SPLINE
SPL {X  -159.452, Y  +378.767, Z    +0.000, E1   +11.887, E3 +105762.657}
SPL {X  -159.840, Y  +384.856, Z    +0.000, E1    +7.126, E3 +105781.629}
SPL {X  -159.991, Y  +390.336, Z    +0.000, E1    +2.803, E3 +105795.451}
SPL {X  -160.000, Y  +403.532, Z    +0.000, E1    -6.523, E3 +105813.172}
SPL {X  -160.000, Y  +409.023, Z    +0.000, E1   -10.003, E3 +105823.946}
SPL {X  -160.000, Y  +418.032, Z    +0.000, E1   -14.569, E3 +105848.805}
SPL {X  -160.000, Y  +420.561, Z    +0.000, E1   -14.816, E3 +105866.285}
SPL {X  -160.000, Y  +422.801, Z    +0.000, E1   -14.823, E3 +105884.233}
SPL {X  -160.000, Y  +425.518, Z    +0.000, E1   -14.845, E3 +105906.008}
SPL {X  -160.000, Y  +428.688, Z    +0.000, E1   -14.854, E3 +105931.416}
SPL {X  -160.000, Y  +431.971, Z    +0.000, E1   -14.849, E3 +105957.885}
SPL {X  -160.000, Y  +435.345, Z    +0.000, E1   -14.857, E3 +105984.935}
SPL {X  -160.000, Y  +438.732, Z    +0.000, E1   -14.858, E3 +106012.083}
SPL {X  -160.000, Y  +441.925, Z    +0.000, E1   -14.848, E3 +106037.754}
SPL {X  -160.000, Y  +444.299, Z    +0.000, E1   -14.809, E3 +106056.938}
SPL {X  -160.000, Y  +446.229, Z    +0.000, E1   -14.820, E3 +106072.357}
SPL {X  -160.000, Y  +448.987, Z    +0.000, E1   -14.868, E3 +106094.294}
SPL {X  -160.000, Y  +452.351, Z    +0.000, E1   -14.871, E3 +106121.270}
SPL {X  -160.000, Y  +455.709, Z    +0.000, E1   -14.880, E3 +106148.084}
SPL {X  -160.000, Y  +458.189, Z    +0.000, E1   -14.832, E3 +106168.086}
SPL {X  -160.000, Y  +459.885, Z    +0.000, E1   -14.825, E3 +106181.757}
SPL {X  -160.000, Y  +462.438, Z    +0.000, E1   -14.868, E3 +106202.167}
SPL {X  -160.000, Y  +465.575, Z    +0.000, E1   -14.849, E3 +106227.475}
SPL {X  -160.000, Y  +468.581, Z    +0.000, E1   -14.841, E3 +106251.707}
SPL {X  -160.000, Y  +471.795, Z    +0.000, E1   -14.854, E3 +106277.495}
SPL {X  -160.000, Y  +475.138, Z    +0.000, E1   -14.853, E3 +106304.345}
SPL {X  -160.000, Y  +477.981, Z    +0.000, E1   -14.823, E3 +106327.265}
SPL {X  -160.000, Y  +480.658, Z    +0.000, E1   -14.835, E3 +106348.741}
SPL {X  -160.000, Y  +483.534, Z    +0.000, E1   -14.838, E3 +106371.836}
SPL {X  -160.000, Y  +486.226, Z    +0.000, E1   -14.823, E3 +106393.501}
SPL {X  -160.000, Y  +488.751, Z    +0.000, E1   -14.827, E3 +106413.774}
SPL {X  -160.000, Y  +491.612, Z    +0.000, E1   -14.844, E3 +106436.696}
SPL {X  -160.000, Y  +494.417, Z    +0.000, E1   -14.827, E3 +106459.287}
SPL {X  -160.000, Y  +496.961, Z    +0.000, E1   -14.824, E3 +106479.731}
SPL {X  -160.000, Y  +499.610, Z    +0.000, E1   -14.830, E3 +106501.004}
SPL {X  -160.000, Y  +502.268, Z    +0.000, E1   -14.832, E3 +106522.273}
SPL {X  -160.000, Y  +505.041, Z    +0.000, E1   -14.849, E3 +106544.435}
SPL {X  -160.000, Y  +507.743, Z    +0.000, E1   -14.842, E3 +106566.059}
SPL {X  -160.000, Y  +510.437, Z    +0.000, E1   -14.860, E3 +106587.573}
SPL {X  -160.000, Y  +513.179, Z    +0.000, E1   -14.849, E3 +106609.620}
SPL {X  -160.000, Y  +515.613, Z    +0.000, E1   -14.829, E3 +106629.291}
SPL {X  -160.000, Y  +518.188, Z    +0.000, E1   -14.845, E3 +106649.920}
SPL {X  -160.000, Y  +520.790, Z    +0.000, E1   -14.839, E3 +106670.749}
SPL {X  -160.000, Y  +523.469, Z    +0.000, E1   -14.855, E3 +106692.197}
SPL {X  -160.000, Y  +526.403, Z    +0.000, E1   -14.858, E3 +106715.734}
SPL {X  -160.000, Y  +529.266, Z    +0.000, E1   -14.848, E3 +106738.741}
SPL {X  -160.000, Y  +531.688, Z    +0.000, E1   -14.826, E3 +106758.291}
SPL {X  -160.000, Y  +534.214, Z    +0.000, E1   -14.841, E3 +106778.554}
SPL {X  -160.000, Y  +537.002, Z    +0.000, E1   -14.839, E3 +106800.972}
SPL {X  -160.000, Y  +539.729, Z    +0.000, E1   -14.840, E3 +106822.783}
SPL {X  -160.000, Y  +542.408, Z    +0.000, E1   -14.839, E3 +106844.336}
SPL {X  -160.000, Y  +545.014, Z    +0.000, E1   -14.831, E3 +106865.282}
SPL {X  -160.000, Y  +547.659, Z    +0.000, E1   -14.839, E3 +106886.496}
SPL {X  -160.000, Y  +550.215, Z    +0.000, E1   -14.827, E3 +106907.061}
SPL {X  -160.000, Y  +552.762, Z    +0.000, E1   -14.836, E3 +106927.479}
SPL {X  -160.000, Y  +555.331, Z    +0.000, E1   -14.837, E3 +106948.020}
SPL {X  -160.000, Y  +558.235, Z    +0.000, E1   -14.869, E3 +106971.184}
SPL {X  -160.000, Y  +561.088, Z    +0.000, E1   -14.848, E3 +106994.102}
SPL {X  -160.000, Y  +563.693, Z    +0.000, E1   -14.852, E3 +107014.963}
SPL {X  -160.000, Y  +566.560, Z    +0.000, E1   -14.865, E3 +107037.941}
SPL {X  -160.000, Y  +569.305, Z    +0.000, E1   -14.848, E3 +107059.969}
SPL {X  -160.000, Y  +571.769, Z    +0.000, E1   -14.852, E3 +107079.715}
SPL {X  -160.000, Y  +574.366, Z    +0.000, E1   -14.855, E3 +107100.502}
SPL {X  -160.000, Y  +577.037, Z    +0.000, E1   -14.859, E3 +107121.901}
SPL {X  -160.000, Y  +579.855, Z    +0.000, E1   -14.869, E3 +107144.429}
SPL {X  -160.000, Y  +582.456, Z    +0.000, E1   -14.854, E3 +107165.289}
SPL {X  -160.000, Y  +585.083, Z    +0.000, E1   -14.866, E3 +107186.338}
SPL {X  -160.000, Y  +587.675, Z    +0.000, E1   -14.853, E3 +107207.129}
SPL {X  -160.000, Y  +590.216, Z    +0.000, E1   -14.864, E3 +107227.448}
SPL {X  -160.000, Y  +592.848, Z    +0.000, E1   -14.865, E3 +107248.500}
SPL {X  -160.000, Y  +595.342, Z    +0.000, E1   -14.848, E3 +107268.677}
SPL {X  -160.000, Y  +597.995, Z    +0.000, E1   -14.848, E3 +107290.017}
SPL {X  -160.000, Y  +600.731, Z    +0.000, E1   -14.846, E3 +107311.969}
SPL {X  -160.000, Y  +603.404, Z    +0.000, E1   -14.846, E3 +107333.404}
SPL {X  -160.000, Y  +605.923, Z    +0.000, E1   -14.838, E3 +107353.645}
SPL {X  -160.000, Y  +608.492, Z    +0.000, E1   -14.846, E3 +107374.249}
SPL {X  -160.000, Y  +611.345, Z    +0.000, E1   -14.856, E3 +107397.107}
SPL {X  -160.000, Y  +614.087, Z    +0.000, E1   -14.839, E3 +107419.166}
SPL {X  -160.000, Y  +616.566, Z    +0.000, E1   -14.839, E3 +107439.060}
SPL {X  -160.000, Y  +619.350, Z    +0.000, E1   -14.855, E3 +107461.348}
SPL {X  -160.000, Y  +622.198, Z    +0.000, E1   -14.846, E3 +107484.233}
SPL {X  -160.000, Y  +624.642, Z    +0.000, E1   -14.829, E3 +107503.905}
SPL {X  -160.000, Y  +627.119, Z    +0.000, E1   -14.843, E3 +107523.745}
SPL {X  -160.000, Y  +629.682, Z    +0.000, E1   -14.838, E3 +107544.314}
SPL {X  -160.000, Y  +632.223, Z    +0.000, E1   -14.841, E3 +107564.705}
SPL {X  -160.000, Y  +634.941, Z    +0.000, E1   -14.846, E3 +107586.503}
SPL {X  -160.000, Y  +637.723, Z    +0.000, E1   -14.844, E3 +107608.847}
SPL {X  -160.000, Y  +640.315, Z    +0.000, E1   -14.836, E3 +107629.645}
SPL {X  -160.000, Y  +643.085, Z    +0.000, E1   -14.865, E3 +107651.696}
SPL {X  -160.000, Y  +645.845, Z    +0.000, E1   -14.848, E3 +107673.884}
SPL {X  -160.000, Y  +648.229, Z    +0.000, E1   -14.834, E3 +107693.094}
SPL {X  -160.000, Y  +650.656, Z    +0.000, E1   -14.835, E3 +107712.651}
SPL {X  -160.000, Y  +653.134, Z    +0.000, E1   -14.827, E3 +107732.578}
SPL {X  -160.000, Y  +655.670, Z    +0.000, E1   -14.841, E3 +107752.872}
SPL {X  -160.000, Y  +658.349, Z    +0.000, E1   -14.842, E3 +107774.347}
SPL {X  -160.000, Y  +660.936, Z    +0.000, E1   -14.838, E3 +107795.099}
SPL {X  -160.000, Y  +663.567, Z    +0.000, E1   -14.845, E3 +107816.230}
SPL {X  -160.000, Y  +666.216, Z    +0.000, E1   -14.832, E3 +107837.546}
SPL {X  -159.997, Y  +668.731, Z    +0.000, E1   -14.834, E3 +107857.738}
SPL {X  -159.962, Y  +671.176, Z    +0.000, E1   -14.822, E3 +107877.449}
SPL {X  -159.895, Y  +673.507, Z    +0.000, E1   -14.821, E3 +107896.181}
SPL {X  -159.785, Y  +675.985, Z    +0.000, E1   -14.818, E3 +107916.182}
SPL {X  -159.627, Y  +678.622, Z    +0.000, E1   -14.804, E3 +107937.535}
SPL {X  -159.438, Y  +681.094, Z    +0.000, E1   -14.770, E3 +107957.706}
SPL {X  -159.262, Y  +683.054, Z    +0.000, E1   -14.719, E3 +107973.935}
ENDSPLINE

SPLINE
SPL {X  -159.661, Y  +678.114, Z    +0.000, E1    -9.575, E3 +108003.527}
SPL {X  -159.942, Y  +672.020, Z    +0.000, E1    -4.692, E3 +108022.153}
SPL {X  -160.000, Y  +664.971, Z    +0.000, E1    +0.516, E3 +108041.704}
SPL {X  -160.000, Y  +660.032, Z    +0.000, E1    +3.995, E3 +108053.647}
SPL {X  -160.000, Y  +652.280, Z    +0.000, E1    +8.913, E3 +108072.162}
SPL {X  -160.000, Y  +644.147, Z    +0.000, E1   +13.158, E3 +108095.712}
SPL {X  -160.000, Y  +641.594, Z    +0.000, E1   +13.488, E3 +108114.153}
SPL {X  -160.000, Y  +639.799, Z    +0.000, E1   +13.486, E3 +108130.063}
SPL {X  -160.000, Y  +637.896, Z    +0.000, E1   +13.493, E3 +108146.878}
SPL {X  -160.000, Y  +635.832, Z    +0.000, E1   +13.499, E3 +108165.137}
SPL {X  -160.000, Y  +633.839, Z    +0.000, E1   +13.489, E3 +108182.826}
SPL {X  -160.000, Y  +631.625, Z    +0.000, E1   +13.508, E3 +108202.366}
SPL {X  -160.000, Y  +629.417, Z    +0.000, E1   +13.491, E3 +108221.978}
SPL {X  -160.000, Y  +627.180, Z    +0.000, E1   +13.508, E3 +108241.732}
SPL {X  -160.000, Y  +624.970, Z    +0.000, E1   +13.490, E3 +108261.382}
SPL {X  -160.000, Y  +623.020, Z    +0.000, E1   +13.491, E3 +108278.612}
SPL {X  -160.000, Y  +620.888, Z    +0.000, E1   +13.501, E3 +108297.474}
SPL {X  -160.000, Y  +618.790, Z    +0.000, E1   +13.488, E3 +108316.096}
SPL {X  -160.000, Y  +616.631, Z    +0.000, E1   +13.504, E3 +108335.150}
SPL {X  -160.000, Y  +614.230, Z    +0.000, E1   +13.510, E3 +108356.346}
SPL {X  -160.000, Y  +612.132, Z    +0.000, E1   +13.485, E3 +108375.062}
SPL {X  -160.000, Y  +610.405, Z    +0.000, E1   +13.477, E3 +108390.436}
SPL {X  -160.000, Y  +608.437, Z    +0.000, E1   +13.502, E3 +108407.691}
SPL {X  -160.000, Y  +606.281, Z    +0.000, E1   +13.502, E3 +108426.709}
SPL {X  -160.000, Y  +604.124, Z    +0.000, E1   +13.513, E3 +108445.764}
SPL {X  -160.000, Y  +601.878, Z    +0.000, E1   +13.505, E3 +108465.661}
SPL {X  -160.000, Y  +599.648, Z    +0.000, E1   +13.506, E3 +108485.438}
SPL {X  -160.000, Y  +597.673, Z    +0.000, E1   +13.479, E3 +108503.111}
SPL {X  -160.000, Y  +595.601, Z    +0.000, E1   +13.499, E3 +108521.395}
SPL {X  -160.000, Y  +593.187, Z    +0.000, E1   +13.500, E3 +108542.775}
SPL {X  -160.000, Y  +591.079, Z    +0.000, E1   +13.483, E3 +108561.501}
SPL {X  -160.000, Y  +589.151, Z    +0.000, E1   +13.489, E3 +108578.552}
SPL {X  -160.000, Y  +586.908, Z    +0.000, E1   +13.501, E3 +108598.397}
SPL {X  -160.000, Y  +584.660, Z    +0.000, E1   +13.490, E3 +108618.339}
SPL {X  -160.000, Y  +582.409, Z    +0.000, E1   +13.499, E3 +108638.257}
SPL {X  -160.000, Y  +580.150, Z    +0.000, E1   +13.490, E3 +108658.304}
SPL {X  -160.000, Y  +577.953, Z    +0.000, E1   +13.493, E3 +108677.762}
SPL {X  -160.000, Y  +575.630, Z    +0.000, E1   +13.502, E3 +108698.246}
SPL {X  -160.000, Y  +573.418, Z    +0.000, E1   +13.502, E3 +108717.754}
SPL {X  -160.000, Y  +571.226, Z    +0.000, E1   +13.520, E3 +108736.963}
SPL {X  -160.000, Y  +569.166, Z    +0.000, E1   +13.512, E3 +108755.153}
SPL {X  -160.000, Y  +567.275, Z    +0.000, E1   +13.517, E3 +108771.820}
SPL {X  -160.000, Y  +565.259, Z    +0.000, E1   +13.523, E3 +108789.609}
SPL {X  -160.000, Y  +563.305, Z    +0.000, E1   +13.512, E3 +108806.948}
SPL {X  -160.000, Y  +561.240, Z    +0.000, E1   +13.521, E3 +108825.209}
SPL {X  -160.000, Y  +558.881, Z    +0.000, E1   +13.524, E3 +108846.052}
SPL {X  -160.000, Y  +556.697, Z    +0.000, E1   +13.510, E3 +108865.438}
SPL {X  -160.000, Y  +554.624, Z    +0.000, E1   +13.512, E3 +108883.769}
SPL {X  -160.000, Y  +552.465, Z    +0.000, E1   +13.514, E3 +108902.853}
SPL {X  -160.000, Y  +550.315, Z    +0.000, E1   +13.514, E3 +108921.846}
SPL {X  -160.000, Y  +548.056, Z    +0.000, E1   +13.519, E3 +108941.847}
SPL {X  -160.000, Y  +545.826, Z    +0.000, E1   +13.501, E3 +108961.725}
SPL {X  -160.000, Y  +543.677, Z    +0.000, E1   +13.502, E3 +108980.783}
SPL {X  -160.000, Y  +541.664, Z    +0.000, E1   +13.489, E3 +108998.668}
SPL {X  -160.000, Y  +539.659, Z    +0.000, E1   +13.494, E3 +109016.429}
SPL {X  -160.000, Y  +537.370, Z    +0.000, E1   +13.501, E3 +109036.668}
SPL {X  -160.000, Y  +535.056, Z    +0.000, E1   +13.506, E3 +109057.063}
SPL {X  -160.000, Y  +532.975, Z    +0.000, E1   +13.494, E3 +109075.550}
SPL {X  -160.000, Y  +530.925, Z    +0.000, E1   +13.499, E3 +109093.712}
SPL {X  -160.000, Y  +528.768, Z    +0.000, E1   +13.498, E3 +109112.813}
SPL {X  -160.000, Y  +526.547, Z    +0.000, E1   +13.499, E3 +109132.482}
SPL {X  -160.000, Y  +523.964, Z    +0.000, E1   +13.742, E3 +109151.986}
SPL {X  -160.000, Y  +513.971, Z    +0.000, E1   +18.644, E3 +109170.898}
SPL {X  -160.000, Y  +513.562, Z    +0.000, E1   +16.972, E3 +109190.775}
SPL {X  -160.000, Y  +513.358, Z    +0.000, E1   +15.267, E3 +109211.047}
SPL {X  -160.000, Y  +512.244, Z    +0.000, E1   +14.473, E3 +109229.503}
SPL {X  -160.000, Y  +509.675, Z    +0.000, E1   +14.481, E3 +109250.647}
SPL {X  -160.000, Y  +507.162, Z    +0.000, E1   +14.470, E3 +109271.387}
SPL {X  -160.000, Y  +504.735, Z    +0.000, E1   +14.473, E3 +109291.358}
SPL {X  -160.000, Y  +502.261, Z    +0.000, E1   +14.476, E3 +109311.694}
SPL {X  -160.000, Y  +499.798, Z    +0.000, E1   +14.482, E3 +109331.896}
SPL {X  -160.000, Y  +497.435, Z    +0.000, E1   +14.476, E3 +109351.373}
SPL {X  -160.000, Y  +495.089, Z    +0.000, E1   +14.475, E3 +109370.740}
SPL {X  -160.000, Y  +492.764, Z    +0.000, E1   +14.469, E3 +109389.911}
SPL {X  -160.000, Y  +490.292, Z    +0.000, E1   +14.476, E3 +109410.312}
SPL {X  -160.000, Y  +487.641, Z    +0.000, E1   +14.470, E3 +109432.208}
SPL {X  -160.000, Y  +485.054, Z    +0.000, E1   +14.460, E3 +109453.651}
SPL {X  -160.000, Y  +482.421, Z    +0.000, E1   +14.461, E3 +109475.369}
SPL {X  -160.000, Y  +480.000, Z    +0.000, E1   +14.451, E3 +109495.334}
SPL {X  -160.000, Y  +477.551, Z    +0.000, E1   +14.466, E3 +109515.462}
SPL {X  -160.000, Y  +475.253, Z    +0.000, E1   +14.450, E3 +109534.436}
SPL {X  -160.000, Y  +473.070, Z    +0.000, E1   +14.454, E3 +109552.457}
SPL {X  -160.000, Y  +470.603, Z    +0.000, E1   +14.464, E3 +109572.757}
SPL {X  -160.000, Y  +468.243, Z    +0.000, E1   +14.458, E3 +109592.157}
SPL {X  -160.000, Y  +465.791, Z    +0.000, E1   +14.475, E3 +109612.301}
SPL {X  -160.000, Y  +463.103, Z    +0.000, E1   +14.474, E3 +109634.449}
SPL {X  -160.000, Y  +460.743, Z    +0.000, E1   +14.465, E3 +109653.858}
SPL {X  -160.000, Y  +458.292, Z    +0.000, E1   +14.492, E3 +109673.857}
SPL {X  -160.000, Y  +455.874, Z    +0.000, E1   +14.484, E3 +109693.715}
SPL {X  -160.000, Y  +453.555, Z    +0.000, E1   +14.488, E3 +109712.794}
SPL {X  -160.000, Y  +451.093, Z    +0.000, E1   +14.485, E3 +109733.106}
SPL {X  -160.000, Y  +448.700, Z    +0.000, E1   +14.483, E3 +109752.795}
SPL {X  -160.000, Y  +446.277, Z    +0.000, E1   +14.485, E3 +109772.719}
SPL {X  -160.000, Y  +443.879, Z    +0.000, E1   +14.485, E3 +109792.457}
SPL {X  -160.000, Y  +441.447, Z    +0.000, E1   +14.485, E3 +109812.464}
SPL {X  -160.000, Y  +439.006, Z    +0.000, E1   +14.488, E3 +109832.547}
SPL {X  -160.000, Y  +436.311, Z    +0.000, E1   +14.498, E3 +109854.706}
SPL {X  -160.000, Y  +433.559, Z    +0.000, E1   +14.491, E3 +109877.376}
SPL {X  -160.000, Y  +431.162, Z    +0.000, E1   +14.479, E3 +109897.127}
SPL {X  -160.000, Y  +429.152, Z    +0.000, E1   +14.469, E3 +109913.708}
SPL {X  -160.000, Y  +426.863, Z    +0.000, E1   +14.490, E3 +109932.487}
SPL {X  -160.000, Y  +424.653, Z    +0.000, E1   +14.467, E3 +109950.747}
SPL {X  -160.000, Y  +422.337, Z    +0.000, E1   +14.492, E3 +109969.731}
SPL {X  -160.000, Y  +419.639, Z    +0.000, E1   +14.504, E3 +109991.771}
SPL {X  -160.000, Y  +417.127, Z    +0.000, E1   +14.501, E3 +110012.362}
SPL {X  -160.000, Y  +414.849, Z    +0.000, E1   +14.496, E3 +110031.096}
SPL {X  -160.000, Y  +412.396, Z    +0.000, E1   +14.505, E3 +110051.285}
SPL {X  -160.000, Y  +409.815, Z    +0.000, E1   +14.498, E3 +110072.539}
SPL {X  -160.000, Y  +407.614, Z    +0.000, E1   +14.484, E3 +110090.665}
SPL {X  -160.000, Y  +405.406, Z    +0.000, E1   +14.501, E3 +110108.728}
SPL {X  -160.000, Y  +402.958, Z    +0.000, E1   +14.500, E3 +110128.898}
SPL {X  -160.000, Y  +400.690, Z    +0.000, E1   +14.484, E3 +110147.609}
SPL {X  -160.000, Y  +398.391, Z    +0.000, E1   +14.502, E3 +110166.435}
SPL {X  -160.000, Y  +395.999, Z    +0.000, E1   +14.484, E3 +110186.225}
SPL {X  -160.000, Y  +393.685, Z    +0.000, E1   +14.486, E3 +110205.298}
SPL {X  -159.999, Y  +391.313, Z    +0.000, E1   +14.479, E3 +110224.880}
SPL {X  -159.970, Y  +388.900, Z    +0.000, E1   +14.480, E3 +110244.764}
SPL {X  -159.903, Y  +386.417, Z    +0.000, E1   +14.475, E3 +110265.269}
SPL {X  -159.796, Y  +383.921, Z    +0.000, E1   +14.466, E3 +110285.925}
SPL {X  -159.651, Y  +381.443, Z    +0.000, E1   +14.453, E3 +110306.472}
SPL {X  -159.474, Y  +379.042, Z    +0.000, E1   +14.434, E3 +110326.436}
SPL {X  -159.316, Y  +377.219, Z    +0.000, E1   +14.400, E3 +110341.665}
ENDSPLINE

SPLINE
SPL {X  -159.452, Y  +378.767, Z    +0.000, E1   +11.887, E3 +110362.654}
SPL {X  -159.840, Y  +384.856, Z    +0.000, E1    +7.126, E3 +110381.625}
SPL {X  -159.991, Y  +390.336, Z    +0.000, E1    +2.803, E3 +110395.448}
SPL {X  -160.000, Y  +403.532, Z    +0.000, E1    -6.523, E3 +110413.169}
SPL {X  -160.000, Y  +409.023, Z    +0.000, E1   -10.003, E3 +110423.942}
SPL {X  -160.000, Y  +418.032, Z    +0.000, E1   -14.569, E3 +110448.802}
SPL {X  -160.000, Y  +420.561, Z    +0.000, E1   -14.816, E3 +110466.282}
SPL {X  -160.000, Y  +422.801, Z    +0.000, E1   -14.823, E3 +110484.230}
SPL {X  -160.000, Y  +425.518, Z    +0.000, E1   -14.845, E3 +110506.005}
SPL {X  -160.000, Y  +428.688, Z    +0.000, E1   -14.854, E3 +110531.413}
SPL {X  -160.000, Y  +431.971, Z    +0.000, E1   -14.849, E3 +110557.882}
SPL {X  -160.000, Y  +435.345, Z    +0.000, E1   -14.857, E3 +110584.932}
SPL {X  -160.000, Y  +438.732, Z    +0.000, E1   -14.858, E3 +110612.080}
SPL {X  -160.000, Y  +441.925, Z    +0.000, E1   -14.848, E3 +110637.751}
SPL {X  -160.000, Y  +444.299, Z    +0.000, E1   -14.809, E3 +110656.935}
SPL {X  -160.000, Y  +446.229, Z    +0.000, E1   -14.820, E3 +110672.354}
SPL {X  -160.000, Y  +448.987, Z    +0.000, E1   -14.868, E3 +110694.291}
SPL {X  -160.000, Y  +452.351, Z    +0.000, E1   -14.871, E3 +110721.267}
SPL {X  -160.000, Y  +455.709, Z    +0.000, E1   -14.880, E3 +110748.081}
SPL {X  -160.000, Y  +458.189, Z    +0.000, E1   -14.832, E3 +110768.083}
SPL {X  -160.000, Y  +459.885, Z    +0.000, E1   -14.825, E3 +110781.753}
SPL {X  -160.000, Y  +462.438, Z    +0.000, E1   -14.868, E3 +110802.163}
SPL {X  -160.000, Y  +465.575, Z    +0.000, E1   -14.849, E3 +110827.472}
SPL {X  -160.000, Y  +468.581, Z    +0.000, E1   -14.841, E3 +110851.704}
SPL {X  -160.000, Y  +471.795, Z    +0.000, E1   -14.854, E3 +110877.491}
SPL {X  -160.000, Y  +475.138, Z    +0.000, E1   -14.853, E3 +110904.342}
SPL {X  -160.000, Y  +477.981, Z    +0.000, E1   -14.823, E3 +110927.262}
SPL {X  -160.000, Y  +480.658, Z    +0.000, E1   -14.835, E3 +110948.738}
SPL {X  -160.000, Y  +483.534, Z    +0.000, E1   -14.838, E3 +110971.833}
SPL {X  -160.000, Y  +486.226, Z    +0.000, E1   -14.823, E3 +110993.498}
SPL {X  -160.000, Y  +488.751, Z    +0.000, E1   -14.827, E3 +111013.770}
SPL {X  -160.000, Y  +491.612, Z    +0.000, E1   -14.844, E3 +111036.693}
SPL {X  -160.000, Y  +494.417, Z    +0.000, E1   -14.827, E3 +111059.284}
SPL {X  -160.000, Y  +496.961, Z    +0.000, E1   -14.824, E3 +111079.728}
SPL {X  -160.000, Y  +499.610, Z    +0.000, E1   -14.830, E3 +111101.000}
SPL {X  -160.000, Y  +502.268, Z    +0.000, E1   -14.832, E3 +111122.270}
SPL {X  -160.000, Y  +505.041, Z    +0.000, E1   -14.849, E3 +111144.432}
SPL {X  -160.000, Y  +507.743, Z    +0.000, E1   -14.842, E3 +111166.056}
SPL {X  -160.000, Y  +510.437, Z    +0.000, E1   -14.860, E3 +111187.570}
SPL {X  -160.000, Y  +513.179, Z    +0.000, E1   -14.849, E3 +111209.617}
SPL {X  -160.000, Y  +515.613, Z    +0.000, E1   -14.829, E3 +111229.288}
SPL {X  -160.000, Y  +518.188, Z    +0.000, E1   -14.845, E3 +111249.917}
SPL {X  -160.000, Y  +520.790, Z    +0.000, E1   -14.839, E3 +111270.746}
SPL {X  -160.000, Y  +523.469, Z    +0.000, E1   -14.855, E3 +111292.194}
SPL {X  -160.000, Y  +526.403, Z    +0.000, E1   -14.858, E3 +111315.730}
SPL {X  -160.000, Y  +529.266, Z    +0.000, E1   -14.848, E3 +111338.738}
SPL {X  -160.000, Y  +531.688, Z    +0.000, E1   -14.826, E3 +111358.287}
SPL {X  -160.000, Y  +534.214, Z    +0.000, E1   -14.841, E3 +111378.550}
SPL {X  -160.000, Y  +537.002, Z    +0.000, E1   -14.839, E3 +111400.969}
SPL {X  -160.000, Y  +539.729, Z    +0.000, E1   -14.840, E3 +111422.780}
SPL {X  -160.000, Y  +542.408, Z    +0.000, E1   -14.839, E3 +111444.333}
SPL {X  -160.000, Y  +545.014, Z    +0.000, E1   -14.831, E3 +111465.278}
SPL {X  -160.000, Y  +547.659, Z    +0.000, E1   -14.839, E3 +111486.493}
SPL {X  -160.000, Y  +550.215, Z    +0.000, E1   -14.827, E3 +111507.058}
SPL {X  -160.000, Y  +552.762, Z    +0.000, E1   -14.836, E3 +111527.476}
SPL {X  -160.000, Y  +555.331, Z    +0.000, E1   -14.837, E3 +111548.017}
SPL {X  -160.000, Y  +558.235, Z    +0.000, E1   -14.869, E3 +111571.181}
SPL {X  -160.000, Y  +561.088, Z    +0.000, E1   -14.848, E3 +111594.099}
SPL {X  -160.000, Y  +563.693, Z    +0.000, E1   -14.852, E3 +111614.960}
SPL {X  -160.000, Y  +566.560, Z    +0.000, E1   -14.865, E3 +111637.937}
SPL {X  -160.000, Y  +569.305, Z    +0.000, E1   -14.848, E3 +111659.966}
SPL {X  -160.000, Y  +571.769, Z    +0.000, E1   -14.852, E3 +111679.712}
SPL {X  -160.000, Y  +574.366, Z    +0.000, E1   -14.855, E3 +111700.499}
SPL {X  -160.000, Y  +577.037, Z    +0.000, E1   -14.859, E3 +111721.898}
SPL {X  -160.000, Y  +579.855, Z    +0.000, E1   -14.869, E3 +111744.425}
SPL {X  -160.000, Y  +582.456, Z    +0.000, E1   -14.854, E3 +111765.285}
SPL {X  -160.000, Y  +585.083, Z    +0.000, E1   -14.866, E3 +111786.335}
SPL {X  -160.000, Y  +587.675, Z    +0.000, E1   -14.853, E3 +111807.126}
SPL {X  -160.000, Y  +590.216, Z    +0.000, E1   -14.864, E3 +111827.445}
SPL {X  -160.000, Y  +592.848, Z    +0.000, E1   -14.865, E3 +111848.496}
SPL {X  -160.000, Y  +595.342, Z    +0.000, E1   -14.848, E3 +111868.674}
SPL {X  -160.000, Y  +597.995, Z    +0.000, E1   -14.848, E3 +111890.014}
SPL {X  -160.000, Y  +600.731, Z    +0.000, E1   -14.846, E3 +111911.965}
SPL {X  -160.000, Y  +603.404, Z    +0.000, E1   -14.846, E3 +111933.401}
SPL {X  -160.000, Y  +605.923, Z    +0.000, E1   -14.838, E3 +111953.642}
SPL {X  -160.000, Y  +608.492, Z    +0.000, E1   -14.846, E3 +111974.246}
SPL {X  -160.000, Y  +611.345, Z    +0.000, E1   -14.856, E3 +111997.104}
SPL {X  -160.000, Y  +614.087, Z    +0.000, E1   -14.839, E3 +112019.163}
SPL {X  -160.000, Y  +616.566, Z    +0.000, E1   -14.839, E3 +112039.057}
SPL {X  -160.000, Y  +619.350, Z    +0.000, E1   -14.855, E3 +112061.345}
SPL {X  -160.000, Y  +622.198, Z    +0.000, E1   -14.846, E3 +112084.230}
SPL {X  -160.000, Y  +624.642, Z    +0.000, E1   -14.829, E3 +112103.902}
SPL {X  -160.000, Y  +627.119, Z    +0.000, E1   -14.843, E3 +112123.742}
SPL {X  -160.000, Y  +629.682, Z    +0.000, E1   -14.838, E3 +112144.311}
SPL {X  -160.000, Y  +632.223, Z    +0.000, E1   -14.841, E3 +112164.702}
SPL {X  -160.000, Y  +634.941, Z    +0.000, E1   -14.846, E3 +112186.500}
SPL {X  -160.000, Y  +637.723, Z    +0.000, E1   -14.844, E3 +112208.844}
SPL {X  -160.000, Y  +640.315, Z    +0.000, E1   -14.836, E3 +112229.642}
SPL {X  -160.000, Y  +643.085, Z    +0.000, E1   -14.865, E3 +112251.693}
SPL {X  -160.000, Y  +645.845, Z    +0.000, E1   -14.848, E3 +112273.881}
SPL {X  -160.000, Y  +648.229, Z    +0.000, E1   -14.834, E3 +112293.091}
SPL {X  -160.000, Y  +650.656, Z    +0.000, E1   -14.835, E3 +112312.647}
SPL {X  -160.000, Y  +653.134, Z    +0.000, E1   -14.827, E3 +112332.574}
SPL {X  -160.000, Y  +655.670, Z    +0.000, E1   -14.841, E3 +112352.869}
SPL {X  -160.000, Y  +658.349, Z    +0.000, E1   -14.842, E3 +112374.344}
SPL {X  -160.000, Y  +660.936, Z    +0.000, E1   -14.838, E3 +112395.096}
SPL {X  -160.000, Y  +663.567, Z    +0.000, E1   -14.845, E3 +112416.226}
SPL {X  -160.000, Y  +666.216, Z    +0.000, E1   -14.832, E3 +112437.543}
SPL {X  -159.997, Y  +668.731, Z    +0.000, E1   -14.834, E3 +112457.735}
SPL {X  -159.962, Y  +671.176, Z    +0.000, E1   -14.822, E3 +112477.446}
SPL {X  -159.895, Y  +673.507, Z    +0.000, E1   -14.821, E3 +112496.177}
SPL {X  -159.785, Y  +675.985, Z    +0.000, E1   -14.818, E3 +112516.179}
SPL {X  -159.627, Y  +678.622, Z    +0.000, E1   -14.804, E3 +112537.532}
SPL {X  -159.438, Y  +681.094, Z    +0.000, E1   -14.770, E3 +112557.703}
SPL {X  -159.262, Y  +683.054, Z    +0.000, E1   -14.719, E3 +112573.931}
ENDSPLINE

SPLINE
SPL {X  -159.661, Y  +678.114, Z    +0.000, E1    -9.575, E3 +112603.523}
SPL {X  -159.942, Y  +672.020, Z    +0.000, E1    -4.692, E3 +112622.150}
SPL {X  -160.000, Y  +664.971, Z    +0.000, E1    +0.516, E3 +112641.700}
SPL {X  -160.000, Y  +660.032, Z    +0.000, E1    +3.995, E3 +112653.643}
SPL {X  -160.000, Y  +652.280, Z    +0.000, E1    +8.913, E3 +112672.158}
SPL {X  -160.000, Y  +644.147, Z    +0.000, E1   +13.158, E3 +112695.709}
SPL {X  -160.000, Y  +641.594, Z    +0.000, E1   +13.488, E3 +112714.150}
SPL {X  -160.000, Y  +639.799, Z    +0.000, E1   +13.486, E3 +112730.060}
SPL {X  -160.000, Y  +637.896, Z    +0.000, E1   +13.493, E3 +112746.875}
SPL {X  -160.000, Y  +635.832, Z    +0.000, E1   +13.499, E3 +112765.134}
SPL {X  -160.000, Y  +633.839, Z    +0.000, E1   +13.489, E3 +112782.822}
SPL {X  -160.000, Y  +631.625, Z    +0.000, E1   +13.508, E3 +112802.363}
SPL {X  -160.000, Y  +629.417, Z    +0.000, E1   +13.491, E3 +112821.975}
SPL {X  -160.000, Y  +627.180, Z    +0.000, E1   +13.508, E3 +112841.729}
SPL {X  -160.000, Y  +624.970, Z    +0.000, E1   +13.490, E3 +112861.379}
SPL {X  -160.000, Y  +623.020, Z    +0.000, E1   +13.491, E3 +112878.608}
SPL {X  -160.000, Y  +620.888, Z    +0.000, E1   +13.501, E3 +112897.471}
SPL {X  -160.000, Y  +618.790, Z    +0.000, E1   +13.488, E3 +112916.093}
SPL {X  -160.000, Y  +616.631, Z    +0.000, E1   +13.504, E3 +112935.147}
SPL {X  -160.000, Y  +614.230, Z    +0.000, E1   +13.510, E3 +112956.343}
SPL {X  -160.000, Y  +612.132, Z    +0.000, E1   +13.485, E3 +112975.059}
SPL {X  -160.000, Y  +610.405, Z    +0.000, E1   +13.477, E3 +112990.432}
SPL {X  -160.000, Y  +608.437, Z    +0.000, E1   +13.502, E3 +113007.688}
SPL {X  -160.000, Y  +606.281, Z    +0.000, E1   +13.502, E3 +113026.705}
SPL {X  -160.000, Y  +604.124, Z    +0.000, E1   +13.513, E3 +113045.761}
SPL {X  -160.000, Y  +601.878, Z    +0.000, E1   +13.505, E3 +113065.658}
SPL {X  -160.000, Y  +599.648, Z    +0.000, E1   +13.506, E3 +113085.435}
SPL {X  -160.000, Y  +597.673, Z    +0.000, E1   +13.479, E3 +113103.108}
SPL {X  -160.000, Y  +595.601, Z    +0.000, E1   +13.499, E3 +113121.391}
SPL {X  -160.000, Y  +593.187, Z    +0.000, E1   +13.500, E3 +113142.771}
SPL {X  -160.000, Y  +591.079, Z    +0.000, E1   +13.483, E3 +113161.498}
SPL {X  -160.000, Y  +589.151, Z    +0.000, E1   +13.489, E3 +113178.549}
SPL {X  -160.000, Y  +586.908, Z    +0.000, E1   +13.501, E3 +113198.394}
SPL {X  -160.000, Y  +584.660, Z    +0.000, E1   +13.490, E3 +113218.336}
SPL {X  -160.000, Y  +582.409, Z    +0.000, E1   +13.499, E3 +113238.254}
SPL {X  -160.000, Y  +580.150, Z    +0.000, E1   +13.490, E3 +113258.300}
SPL {X  -160.000, Y  +577.953, Z    +0.000, E1   +13.493, E3 +113277.759}
SPL {X  -160.000, Y  +575.630, Z    +0.000, E1   +13.502, E3 +113298.243}
SPL {X  -160.000, Y  +573.418, Z    +0.000, E1   +13.502, E3 +113317.751}
SPL {X  -160.000, Y  +571.226, Z    +0.000, E1   +13.520, E3 +113336.959}
SPL {X  -160.000, Y  +569.166, Z    +0.000, E1   +13.512, E3 +113355.150}
SPL {X  -160.000, Y  +567.275, Z    +0.000, E1   +13.517, E3 +113371.817}
SPL {X  -160.000, Y  +565.259, Z    +0.000, E1   +13.523, E3 +113389.606}
SPL {X  -160.000, Y  +563.305, Z    +0.000, E1   +13.512, E3 +113406.945}
SPL {X  -160.000, Y  +561.240, Z    +0.000, E1   +13.521, E3 +113425.206}
SPL {X  -160.000, Y  +558.881, Z    +0.000, E1   +13.524, E3 +113446.049}
SPL {X  -160.000, Y  +556.697, Z    +0.000, E1   +13.510, E3 +113465.434}
SPL {X  -160.000, Y  +554.624, Z    +0.000, E1   +13.512, E3 +113483.765}
SPL {X  -160.000, Y  +552.465, Z    +0.000, E1   +13.514, E3 +113502.850}
SPL {X  -160.000, Y  +550.315, Z    +0.000, E1   +13.514, E3 +113521.843}
SPL {X  -160.000, Y  +548.056, Z    +0.000, E1   +13.519, E3 +113541.844}
SPL {X  -160.000, Y  +545.826, Z    +0.000, E1   +13.501, E3 +113561.722}
SPL {X  -160.000, Y  +543.677, Z    +0.000, E1   +13.502, E3 +113580.780}
SPL {X  -160.000, Y  +541.664, Z    +0.000, E1   +13.489, E3 +113598.665}
SPL {X  -160.000, Y  +539.659, Z    +0.000, E1   +13.494, E3 +113616.425}
SPL {X  -160.000, Y  +537.370, Z    +0.000, E1   +13.501, E3 +113636.664}
SPL {X  -160.000, Y  +535.056, Z    +0.000, E1   +13.506, E3 +113657.060}
SPL {X  -160.000, Y  +532.975, Z    +0.000, E1   +13.494, E3 +113675.547}
SPL {X  -160.000, Y  +530.925, Z    +0.000, E1   +13.499, E3 +113693.708}
SPL {X  -160.000, Y  +528.768, Z    +0.000, E1   +13.498, E3 +113712.810}
SPL {X  -160.000, Y  +526.547, Z    +0.000, E1   +13.499, E3 +113732.478}
SPL {X  -160.000, Y  +523.964, Z    +0.000, E1   +13.742, E3 +113751.983}
SPL {X  -160.000, Y  +513.971, Z    +0.000, E1   +18.644, E3 +113770.895}
SPL {X  -160.000, Y  +513.562, Z    +0.000, E1   +16.972, E3 +113790.772}
SPL {X  -160.000, Y  +513.358, Z    +0.000, E1   +15.267, E3 +113811.044}
SPL {X  -160.000, Y  +512.244, Z    +0.000, E1   +14.473, E3 +113829.500}
SPL {X  -160.000, Y  +509.675, Z    +0.000, E1   +14.481, E3 +113850.643}
SPL {X  -160.000, Y  +507.162, Z    +0.000, E1   +14.470, E3 +113871.383}
SPL {X  -160.000, Y  +504.735, Z    +0.000, E1   +14.473, E3 +113891.355}
SPL {X  -160.000, Y  +502.261, Z    +0.000, E1   +14.476, E3 +113911.691}
SPL {X  -160.000, Y  +499.798, Z    +0.000, E1   +14.482, E3 +113931.893}
SPL {X  -160.000, Y  +497.435, Z    +0.000, E1   +14.476, E3 +113951.370}
SPL {X  -160.000, Y  +495.089, Z    +0.000, E1   +14.475, E3 +113970.737}
SPL {X  -160.000, Y  +492.764, Z    +0.000, E1   +14.469, E3 +113989.908}
SPL {X  -160.000, Y  +490.292, Z    +0.000, E1   +14.476, E3 +114010.309}
SPL {X  -160.000, Y  +487.641, Z    +0.000, E1   +14.470, E3 +114032.205}
SPL {X  -160.000, Y  +485.054, Z    +0.000, E1   +14.460, E3 +114053.648}
SPL {X  -160.000, Y  +482.421, Z    +0.000, E1   +14.461, E3 +114075.366}
SPL {X  -160.000, Y  +480.000, Z    +0.000, E1   +14.451, E3 +114095.330}
SPL {X  -160.000, Y  +477.551, Z    +0.000, E1   +14.466, E3 +114115.459}
SPL {X  -160.000, Y  +475.253, Z    +0.000, E1   +14.450, E3 +114134.433}
SPL {X  -160.000, Y  +473.070, Z    +0.000, E1   +14.454, E3 +114152.454}
SPL {X  -160.000, Y  +470.603, Z    +0.000, E1   +14.464, E3 +114172.754}
SPL {X  -160.000, Y  +468.243, Z    +0.000, E1   +14.458, E3 +114192.153}
SPL {X  -160.000, Y  +465.791, Z    +0.000, E1   +14.475, E3 +114212.298}
SPL {X  -160.000, Y  +463.103, Z    +0.000, E1   +14.474, E3 +114234.446}
SPL {X  -160.000, Y  +460.743, Z    +0.000, E1   +14.465, E3 +114253.855}
SPL {X  -160.000, Y  +458.292, Z    +0.000, E1   +14.492, E3 +114273.854}
SPL {X  -160.000, Y  +455.874, Z    +0.000, E1   +14.484, E3 +114293.711}
SPL {X  -160.000, Y  +453.555, Z    +0.000, E1   +14.488, E3 +114312.791}
SPL {X  -160.000, Y  +451.093, Z    +0.000, E1   +14.485, E3 +114333.103}
SPL {X  -160.000, Y  +448.700, Z    +0.000, E1   +14.483, E3 +114352.792}
SPL {X  -160.000, Y  +446.277, Z    +0.000, E1   +14.485, E3 +114372.716}
SPL {X  -160.000, Y  +443.879, Z    +0.000, E1   +14.485, E3 +114392.454}
SPL {X  -160.000, Y  +441.447, Z    +0.000, E1   +14.485, E3 +114412.461}
SPL {X  -160.000, Y  +439.006, Z    +0.000, E1   +14.488, E3 +114432.544}
SPL {X  -160.000, Y  +436.311, Z    +0.000, E1   +14.498, E3 +114454.703}
SPL {X  -160.000, Y  +433.559, Z    +0.000, E1   +14.491, E3 +114477.373}
SPL {X  -160.000, Y  +431.162, Z    +0.000, E1   +14.479, E3 +114497.124}
SPL {X  -160.000, Y  +429.152, Z    +0.000, E1   +14.469, E3 +114513.705}
SPL {X  -160.000, Y  +426.863, Z    +0.000, E1   +14.490, E3 +114532.484}
SPL {X  -160.000, Y  +424.653, Z    +0.000, E1   +14.467, E3 +114550.744}
SPL {X  -160.000, Y  +422.337, Z    +0.000, E1   +14.492, E3 +114569.728}
SPL {X  -160.000, Y  +419.639, Z    +0.000, E1   +14.504, E3 +114591.768}
SPL {X  -160.000, Y  +417.127, Z    +0.000, E1   +14.501, E3 +114612.359}
SPL {X  -160.000, Y  +414.849, Z    +0.000, E1   +14.496, E3 +114631.093}
SPL {X  -160.000, Y  +412.396, Z    +0.000, E1   +14.505, E3 +114651.282}
SPL {X  -160.000, Y  +409.815, Z    +0.000, E1   +14.498, E3 +114672.536}
SPL {X  -160.000, Y  +407.614, Z    +0.000, E1   +14.484, E3 +114690.661}
SPL {X  -160.000, Y  +405.406, Z    +0.000, E1   +14.501, E3 +114708.724}
SPL {X  -160.000, Y  +402.958, Z    +0.000, E1   +14.500, E3 +114728.895}
SPL {X  -160.000, Y  +400.690, Z    +0.000, E1   +14.484, E3 +114747.606}
SPL {X  -160.000, Y  +398.391, Z    +0.000, E1   +14.502, E3 +114766.432}
SPL {X  -160.000, Y  +395.999, Z    +0.000, E1   +14.484, E3 +114786.222}
SPL {X  -160.000, Y  +393.685, Z    +0.000, E1   +14.486, E3 +114805.294}
SPL {X  -159.999, Y  +391.313, Z    +0.000, E1   +14.479, E3 +114824.876}
SPL {X  -159.970, Y  +388.900, Z    +0.000, E1   +14.480, E3 +114844.761}
SPL {X  -159.903, Y  +386.417, Z    +0.000, E1   +14.475, E3 +114865.266}
SPL {X  -159.796, Y  +383.921, Z    +0.000, E1   +14.466, E3 +114885.921}
SPL {X  -159.651, Y  +381.443, Z    +0.000, E1   +14.453, E3 +114906.469}
SPL {X  -159.474, Y  +379.042, Z    +0.000, E1   +14.434, E3 +114926.433}
SPL {X  -159.316, Y  +377.219, Z    +0.000, E1   +14.400, E3 +114941.661}
ENDSPLINE

SPLINE
SPL {X  -159.452, Y  +378.767, Z    +0.000, E1   +11.887, E3 +114962.651}
SPL {X  -159.840, Y  +384.856, Z    +0.000, E1    +7.126, E3 +114981.622}
SPL {X  -159.991, Y  +390.336, Z    +0.000, E1    +2.803, E3 +114995.445}
SPL {X  -160.000, Y  +403.532, Z    +0.000, E1    -6.523, E3 +115013.166}
SPL {X  -160.000, Y  +409.023, Z    +0.000, E1   -10.003, E3 +115023.939}
SPL {X  -160.000, Y  +418.032, Z    +0.000, E1   -14.569, E3 +115048.798}
SPL {X  -160.000, Y  +420.561, Z    +0.000, E1   -14.816, E3 +115066.279}
SPL {X  -160.000, Y  +422.801, Z    +0.000, E1   -14.823, E3 +115084.227}
SPL {X  -160.000, Y  +425.518, Z    +0.000, E1   -14.845, E3 +115106.002}
SPL {X  -160.000, Y  +428.688, Z    +0.000, E1   -14.854, E3 +115131.410}
SPL {X  -160.000, Y  +431.971, Z    +0.000, E1   -14.849, E3 +115157.878}
SPL {X  -160.000, Y  +435.345, Z    +0.000, E1   -14.857, E3 +115184.929}
SPL {X  -160.000, Y  +438.732, Z    +0.000, E1   -14.858, E3 +115212.077}
SPL {X  -160.000, Y  +441.925, Z    +0.000, E1   -14.848, E3 +115237.747}
SPL {X  -160.000, Y  +444.299, Z    +0.000, E1   -14.809, E3 +115256.932}
SPL {X  -160.000, Y  +446.229, Z    +0.000, E1   -14.820, E3 +115272.351}
SPL {X  -160.000, Y  +448.987, Z    +0.000, E1   -14.868, E3 +115294.288}
SPL {X  -160.000, Y  +452.351, Z    +0.000, E1   -14.871, E3 +115321.264}
SPL {X  -160.000, Y  +455.709, Z    +0.000, E1   -14.880, E3 +115348.078}
SPL {X  -160.000, Y  +458.189, Z    +0.000, E1   -14.832, E3 +115368.079}
SPL {X  -160.000, Y  +459.885, Z    +0.000, E1   -14.825, E3 +115381.750}
SPL {X  -160.000, Y  +462.438, Z    +0.000, E1   -14.868, E3 +115402.160}
SPL {X  -160.000, Y  +465.575, Z    +0.000, E1   -14.849, E3 +115427.468}
SPL {X  -160.000, Y  +468.581, Z    +0.000, E1   -14.841, E3 +115451.701}
SPL {X  -160.000, Y  +471.795, Z    +0.000, E1   -14.854, E3 +115477.488}
SPL {X  -160.000, Y  +475.138, Z    +0.000, E1   -14.853, E3 +115504.339}
SPL {X  -160.000, Y  +477.981, Z    +0.000, E1   -14.823, E3 +115527.259}
SPL {X  -160.000, Y  +480.658, Z    +0.000, E1   -14.835, E3 +115548.735}
SPL {X  -160.000, Y  +483.534, Z    +0.000, E1   -14.838, E3 +115571.830}
SPL {X  -160.000, Y  +486.226, Z    +0.000, E1   -14.823, E3 +115593.495}
SPL {X  -160.000, Y  +488.751, Z    +0.000, E1   -14.827, E3 +115613.767}
SPL {X  -160.000, Y  +491.612, Z    +0.000, E1   -14.844, E3 +115636.690}
SPL {X  -160.000, Y  +494.417, Z    +0.000, E1   -14.827, E3 +115659.281}
SPL {X  -160.000, Y  +496.961, Z    +0.000, E1   -14.824, E3 +115679.725}
SPL {X  -160.000, Y  +499.610, Z    +0.000, E1   -14.830, E3 +115700.997}
SPL {X  -160.000, Y  +502.268, Z    +0.000, E1   -14.832, E3 +115722.266}
SPL {X  -160.000, Y  +505.041, Z    +0.000, E1   -14.849, E3 +115744.429}
SPL {X  -160.000, Y  +507.743, Z    +0.000, E1   -14.842, E3 +115766.053}
SPL {X  -160.000, Y  +510.437, Z    +0.000, E1   -14.860, E3 +115787.567}
SPL {X  -160.000, Y  +513.179, Z    +0.000, E1   -14.849, E3 +115809.614}
SPL {X  -160.000, Y  +515.613, Z    +0.000, E1   -14.829, E3 +115829.284}
SPL {X  -160.000, Y  +518.188, Z    +0.000, E1   -14.845, E3 +115849.914}
SPL {X  -160.000, Y  +520.790, Z    +0.000, E1   -14.839, E3 +115870.743}
SPL {X  -160.000, Y  +523.469, Z    +0.000, E1   -14.855, E3 +115892.191}
SPL {X  -160.000, Y  +526.403, Z    +0.000, E1   -14.858, E3 +115915.727}
SPL {X  -160.000, Y  +529.266, Z    +0.000, E1   -14.848, E3 +115938.735}
SPL {X  -160.000, Y  +531.688, Z    +0.000, E1   -14.826, E3 +115958.284}
SPL {X  -160.000, Y  +534.214, Z    +0.000, E1   -14.841, E3 +115978.547}
SPL {X  -160.000, Y  +537.002, Z    +0.000, E1   -14.839, E3 +116000.965}
SPL {X  -160.000, Y  +539.729, Z    +0.000, E1   -14.840, E3 +116022.777}
SPL {X  -160.000, Y  +542.408, Z    +0.000, E1   -14.839, E3 +116044.330}
SPL {X  -160.000, Y  +545.014, Z    +0.000, E1   -14.831, E3 +116065.275}
SPL {X  -160.000, Y  +547.659, Z    +0.000, E1   -14.839, E3 +116086.490}
SPL {X  -160.000, Y  +550.215, Z    +0.000, E1   -14.827, E3 +116107.055}
SPL {X  -160.000, Y  +552.762, Z    +0.000, E1   -14.836, E3 +116127.473}
SPL {X  -160.000, Y  +555.331, Z    +0.000, E1   -14.837, E3 +116148.014}
SPL {X  -160.000, Y  +558.235, Z    +0.000, E1   -14.869, E3 +116171.177}
SPL {X  -160.000, Y  +561.088, Z    +0.000, E1   -14.848, E3 +116194.096}
SPL {X  -160.000, Y  +563.693, Z    +0.000, E1   -14.852, E3 +116214.957}
SPL {X  -160.000, Y  +566.560, Z    +0.000, E1   -14.865, E3 +116237.934}
SPL {X  -160.000, Y  +569.305, Z    +0.000, E1   -14.848, E3 +116259.963}
SPL {X  -160.000, Y  +571.769, Z    +0.000, E1   -14.852, E3 +116279.708}
SPL {X  -160.000, Y  +574.366, Z    +0.000, E1   -14.855, E3 +116300.495}
SPL {X  -160.000, Y  +577.037, Z    +0.000, E1   -14.859, E3 +116321.895}
SPL {X  -160.000, Y  +579.855, Z    +0.000, E1   -14.869, E3 +116344.422}
SPL {X  -160.000, Y  +582.456, Z    +0.000, E1   -14.854, E3 +116365.282}
SPL {X  -160.000, Y  +585.083, Z    +0.000, E1   -14.866, E3 +116386.332}
SPL {X  -160.000, Y  +587.675, Z    +0.000, E1   -14.853, E3 +116407.123}
SPL {X  -160.000, Y  +590.216, Z    +0.000, E1   -14.864, E3 +116427.442}
SPL {X  -160.000, Y  +592.848, Z    +0.000, E1   -14.865, E3 +116448.493}
SPL {X  -160.000, Y  +595.342, Z    +0.000, E1   -14.848, E3 +116468.671}
SPL {X  -160.000, Y  +597.995, Z    +0.000, E1   -14.848, E3 +116490.011}
SPL {X  -160.000, Y  +600.731, Z    +0.000, E1   -14.846, E3 +116511.962}
SPL {X  -160.000, Y  +603.404, Z    +0.000, E1   -14.846, E3 +116533.398}
SPL {X  -160.000, Y  +605.923, Z    +0.000, E1   -14.838, E3 +116553.639}
SPL {X  -160.000, Y  +608.492, Z    +0.000, E1   -14.846, E3 +116574.243}
SPL {X  -160.000, Y  +611.345, Z    +0.000, E1   -14.856, E3 +116597.101}
SPL {X  -160.000, Y  +614.087, Z    +0.000, E1   -14.839, E3 +116619.160}
SPL {X  -160.000, Y  +616.566, Z    +0.000, E1   -14.839, E3 +116639.054}
SPL {X  -160.000, Y  +619.350, Z    +0.000, E1   -14.855, E3 +116661.342}
SPL {X  -160.000, Y  +622.198, Z    +0.000, E1   -14.846, E3 +116684.226}
SPL {X  -160.000, Y  +624.642, Z    +0.000, E1   -14.829, E3 +116703.899}
SPL {X  -160.000, Y  +627.119, Z    +0.000, E1   -14.843, E3 +116723.739}
SPL {X  -160.000, Y  +629.682, Z    +0.000, E1   -14.838, E3 +116744.308}
SPL {X  -160.000, Y  +632.223, Z    +0.000, E1   -14.841, E3 +116764.699}
SPL {X  -160.000, Y  +634.941, Z    +0.000, E1   -14.846, E3 +116786.497}
SPL {X  -160.000, Y  +637.723, Z    +0.000, E1   -14.844, E3 +116808.841}
SPL {X  -160.000, Y  +640.315, Z    +0.000, E1   -14.836, E3 +116829.638}
SPL {X  -160.000, Y  +643.085, Z    +0.000, E1   -14.865, E3 +116851.690}
SPL {X  -160.000, Y  +645.845, Z    +0.000, E1   -14.848, E3 +116873.878}
SPL {X  -160.000, Y  +648.229, Z    +0.000, E1   -14.834, E3 +116893.088}
SPL {X  -160.000, Y  +650.656, Z    +0.000, E1   -14.835, E3 +116912.644}
SPL {X  -160.000, Y  +653.134, Z    +0.000, E1   -14.827, E3 +116932.571}
SPL {X  -160.000, Y  +655.670, Z    +0.000, E1   -14.841, E3 +116952.865}
SPL {X  -160.000, Y  +658.349, Z    +0.000, E1   -14.842, E3 +116974.341}
SPL {X  -160.000, Y  +660.936, Z    +0.000, E1   -14.838, E3 +116995.093}
SPL {X  -160.000, Y  +663.567, Z    +0.000, E1   -14.845, E3 +117016.223}
SPL {X  -160.000, Y  +666.216, Z    +0.000, E1   -14.832, E3 +117037.540}
SPL {X  -159.997, Y  +668.731, Z    +0.000, E1   -14.834, E3 +117057.732}
SPL {X  -159.962, Y  +671.176, Z    +0.000, E1   -14.822, E3 +117077.443}
SPL {X  -159.895, Y  +673.507, Z    +0.000, E1   -14.821, E3 +117096.174}
SPL {X  -159.785, Y  +675.985, Z    +0.000, E1   -14.818, E3 +117116.176}
SPL {X  -159.627, Y  +678.622, Z    +0.000, E1   -14.804, E3 +117137.528}
SPL {X  -159.438, Y  +681.094, Z    +0.000, E1   -14.770, E3 +117157.700}
SPL {X  -159.262, Y  +683.054, Z    +0.000, E1   -14.719, E3 +117173.928}
ENDSPLINE

SPLINE
SPL {X  -159.661, Y  +678.114, Z    +0.000, E1    -9.575, E3 +117203.520}
SPL {X  -159.942, Y  +672.020, Z    +0.000, E1    -4.692, E3 +117222.147}
SPL {X  -160.000, Y  +664.971, Z    +0.000, E1    +0.516, E3 +117241.697}
SPL {X  -160.000, Y  +660.032, Z    +0.000, E1    +3.995, E3 +117253.640}
SPL {X  -160.000, Y  +652.280, Z    +0.000, E1    +8.913, E3 +117272.155}
SPL {X  -160.000, Y  +644.147, Z    +0.000, E1   +13.158, E3 +117295.706}
SPL {X  -160.000, Y  +641.594, Z    +0.000, E1   +13.488, E3 +117314.147}
SPL {X  -160.000, Y  +639.799, Z    +0.000, E1   +13.486, E3 +117330.057}
SPL {X  -160.000, Y  +637.896, Z    +0.000, E1   +13.493, E3 +117346.872}
SPL {X  -160.000, Y  +635.832, Z    +0.000, E1   +13.499, E3 +117365.130}
SPL {X  -160.000, Y  +633.839, Z    +0.000, E1   +13.489, E3 +117382.819}
SPL {X  -160.000, Y  +631.625, Z    +0.000, E1   +13.508, E3 +117402.360}
SPL {X  -160.000, Y  +629.417, Z    +0.000, E1   +13.491, E3 +117421.971}
SPL {X  -160.000, Y  +627.180, Z    +0.000, E1   +13.508, E3 +117441.725}
SPL {X  -160.000, Y  +624.970, Z    +0.000, E1   +13.490, E3 +117461.375}
SPL {X  -160.000, Y  +623.020, Z    +0.000, E1   +13.491, E3 +117478.605}
SPL {X  -160.000, Y  +620.888, Z    +0.000, E1   +13.501, E3 +117497.468}
SPL {X  -160.000, Y  +618.790, Z    +0.000, E1   +13.488, E3 +117516.090}
SPL {X  -160.000, Y  +616.631, Z    +0.000, E1   +13.504, E3 +117535.144}
SPL {X  -160.000, Y  +614.230, Z    +0.000, E1   +13.510, E3 +117556.339}
SPL {X  -160.000, Y  +612.132, Z    +0.000, E1   +13.485, E3 +117575.056}
SPL {X  -160.000, Y  +610.405, Z    +0.000, E1   +13.477, E3 +117590.429}
SPL {X  -160.000, Y  +608.437, Z    +0.000, E1   +13.502, E3 +117607.685}
SPL {X  -160.000, Y  +606.281, Z    +0.000, E1   +13.502, E3 +117626.702}
SPL {X  -160.000, Y  +604.124, Z    +0.000, E1   +13.513, E3 +117645.757}
SPL {X  -160.000, Y  +601.878, Z    +0.000, E1   +13.505, E3 +117665.655}
SPL {X  -160.000, Y  +599.648, Z    +0.000, E1   +13.506, E3 +117685.431}
SPL {X  -160.000, Y  +597.673, Z    +0.000, E1   +13.479, E3 +117703.105}
SPL {X  -160.000, Y  +595.601, Z    +0.000, E1   +13.499, E3 +117721.388}
SPL {X  -160.000, Y  +593.187, Z    +0.000, E1   +13.500, E3 +117742.768}
SPL {X  -160.000, Y  +591.079, Z    +0.000, E1   +13.483, E3 +117761.494}
SPL {X  -160.000, Y  +589.151, Z    +0.000, E1   +13.489, E3 +117778.545}
SPL {X  -160.000, Y  +586.908, Z    +0.000, E1   +13.501, E3 +117798.391}
SPL {X  -160.000, Y  +584.660, Z    +0.000, E1   +13.490, E3 +117818.332}
SPL {X  -160.000, Y  +582.409, Z    +0.000, E1   +13.499, E3 +117838.251}
SPL {X  -160.000, Y  +580.150, Z    +0.000, E1   +13.490, E3 +117858.297}
SPL {X  -160.000, Y  +577.953, Z    +0.000, E1   +13.493, E3 +117877.755}
SPL {X  -160.000, Y  +575.630, Z    +0.000, E1   +13.502, E3 +117898.239}
SPL {X  -160.000, Y  +573.418, Z    +0.000, E1   +13.502, E3 +117917.747}
SPL {X  -160.000, Y  +571.226, Z    +0.000, E1   +13.520, E3 +117936.956}
SPL {X  -160.000, Y  +569.166, Z    +0.000, E1   +13.512, E3 +117955.147}
SPL {X  -160.000, Y  +567.275, Z    +0.000, E1   +13.517, E3 +117971.814}
SPL {X  -160.000, Y  +565.259, Z    +0.000, E1   +13.523, E3 +117989.603}
SPL {X  -160.000, Y  +563.305, Z    +0.000, E1   +13.512, E3 +118006.941}
SPL {X  -160.000, Y  +561.240, Z    +0.000, E1   +13.521, E3 +118025.203}
SPL {X  -160.000, Y  +558.881, Z    +0.000, E1   +13.524, E3 +118046.045}
SPL {X  -160.000, Y  +556.697, Z    +0.000, E1   +13.510, E3 +118065.431}
SPL {X  -160.000, Y  +554.624, Z    +0.000, E1   +13.512, E3 +118083.762}
SPL {X  -160.000, Y  +552.465, Z    +0.000, E1   +13.514, E3 +118102.846}
SPL {X  -160.000, Y  +550.315, Z    +0.000, E1   +13.514, E3 +118121.840}
SPL {X  -160.000, Y  +548.056, Z    +0.000, E1   +13.519, E3 +118141.841}
SPL {X  -160.000, Y  +545.826, Z    +0.000, E1   +13.501, E3 +118161.719}
SPL {X  -160.000, Y  +543.677, Z    +0.000, E1   +13.502, E3 +118180.777}
SPL {X  -160.000, Y  +541.664, Z    +0.000, E1   +13.489, E3 +118198.662}
SPL {X  -160.000, Y  +539.659, Z    +0.000, E1   +13.494, E3 +118216.422}
SPL {X  -160.000, Y  +537.370, Z    +0.000, E1   +13.501, E3 +118236.661}
SPL {X  -160.000, Y  +535.056, Z    +0.000, E1   +13.506, E3 +118257.057}
SPL {X  -160.000, Y  +532.975, Z    +0.000, E1   +13.494, E3 +118275.544}
SPL {X  -160.000, Y  +530.925, Z    +0.000, E1   +13.499, E3 +118293.705}
SPL {X  -160.000, Y  +528.768, Z    +0.000, E1   +13.498, E3 +118312.807}
SPL {X  -160.000, Y  +526.547, Z    +0.000, E1   +13.499, E3 +118332.475}
SPL {X  -160.000, Y  +523.964, Z    +0.000, E1   +13.742, E3 +118351.980}
SPL {X  -160.000, Y  +513.971, Z    +0.000, E1   +18.644, E3 +118370.892}
SPL {X  -160.000, Y  +513.562, Z    +0.000, E1   +16.972, E3 +118390.768}
SPL {X  -160.000, Y  +513.358, Z    +0.000, E1   +15.267, E3 +118411.040}
SPL {X  -160.000, Y  +512.244, Z    +0.000, E1   +14.473, E3 +118429.497}
SPL {X  -160.000, Y  +509.675, Z    +0.000, E1   +14.481, E3 +118450.640}
SPL {X  -160.000, Y  +507.162, Z    +0.000, E1   +14.470, E3 +118471.380}
SPL {X  -160.000, Y  +504.735, Z    +0.000, E1   +14.473, E3 +118491.352}
SPL {X  -160.000, Y  +502.261, Z    +0.000, E1   +14.476, E3 +118511.688}
SPL {X  -160.000, Y  +499.798, Z    +0.000, E1   +14.482, E3 +118531.890}
SPL {X  -160.000, Y  +497.435, Z    +0.000, E1   +14.476, E3 +118551.367}
SPL {X  -160.000, Y  +495.089, Z    +0.000, E1   +14.475, E3 +118570.733}
SPL {X  -160.000, Y  +492.764, Z    +0.000, E1   +14.469, E3 +118589.905}
SPL {X  -160.000, Y  +490.292, Z    +0.000, E1   +14.476, E3 +118610.306}
SPL {X  -160.000, Y  +487.641, Z    +0.000, E1   +14.470, E3 +118632.202}
SPL {X  -160.000, Y  +485.054, Z    +0.000, E1   +14.460, E3 +118653.645}
SPL {X  -160.000, Y  +482.421, Z    +0.000, E1   +14.461, E3 +118675.363}
SPL {X  -160.000, Y  +480.000, Z    +0.000, E1   +14.451, E3 +118695.327}
SPL {X  -160.000, Y  +477.551, Z    +0.000, E1   +14.466, E3 +118715.456}
SPL {X  -160.000, Y  +475.253, Z    +0.000, E1   +14.450, E3 +118734.430}
SPL {X  -160.000, Y  +473.070, Z    +0.000, E1   +14.454, E3 +118752.451}
SPL {X  -160.000, Y  +470.603, Z    +0.000, E1   +14.464, E3 +118772.751}
SPL {X  -160.000, Y  +468.243, Z    +0.000, E1   +14.458, E3 +118792.150}
SPL {X  -160.000, Y  +465.791, Z    +0.000, E1   +14.475, E3 +118812.294}
SPL {X  -160.000, Y  +463.103, Z    +0.000, E1   +14.474, E3 +118834.443}
SPL {X  -160.000, Y  +460.743, Z    +0.000, E1   +14.465, E3 +118853.851}
SPL {X  -160.000, Y  +458.292, Z    +0.000, E1   +14.492, E3 +118873.851}
SPL {X  -160.000, Y  +455.874, Z    +0.000, E1   +14.484, E3 +118893.708}
SPL {X  -160.000, Y  +453.555, Z    +0.000, E1   +14.488, E3 +118912.787}
SPL {X  -160.000, Y  +451.093, Z    +0.000, E1   +14.485, E3 +118933.100}
SPL {X  -160.000, Y  +448.700, Z    +0.000, E1   +14.483, E3 +118952.789}
SPL {X  -160.000, Y  +446.277, Z    +0.000, E1   +14.485, E3 +118972.713}
SPL {X  -160.000, Y  +443.879, Z    +0.000, E1   +14.485, E3 +118992.451}
SPL {X  -160.000, Y  +441.447, Z    +0.000, E1   +14.485, E3 +119012.458}
SPL {X  -160.000, Y  +439.006, Z    +0.000, E1   +14.488, E3 +119032.541}
SPL {X  -160.000, Y  +436.311, Z    +0.000, E1   +14.498, E3 +119054.700}
SPL {X  -160.000, Y  +433.559, Z    +0.000, E1   +14.491, E3 +119077.369}
SPL {X  -160.000, Y  +431.162, Z    +0.000, E1   +14.479, E3 +119097.121}
SPL {X  -160.000, Y  +429.152, Z    +0.000, E1   +14.469, E3 +119113.702}
SPL {X  -160.000, Y  +426.863, Z    +0.000, E1   +14.490, E3 +119132.481}
SPL {X  -160.000, Y  +424.653, Z    +0.000, E1   +14.467, E3 +119150.740}
SPL {X  -160.000, Y  +422.337, Z    +0.000, E1   +14.492, E3 +119169.725}
SPL {X  -160.000, Y  +419.639, Z    +0.000, E1   +14.504, E3 +119191.764}
SPL {X  -160.000, Y  +417.127, Z    +0.000, E1   +14.501, E3 +119212.356}
SPL {X  -160.000, Y  +414.849, Z    +0.000, E1   +14.496, E3 +119231.090}
SPL {X  -160.000, Y  +412.396, Z    +0.000, E1   +14.505, E3 +119251.279}
SPL {X  -160.000, Y  +409.815, Z    +0.000, E1   +14.498, E3 +119272.533}
SPL {X  -160.000, Y  +407.614, Z    +0.000, E1   +14.484, E3 +119290.658}
SPL {X  -160.000, Y  +405.406, Z    +0.000, E1   +14.501, E3 +119308.721}
SPL {X  -160.000, Y  +402.958, Z    +0.000, E1   +14.500, E3 +119328.891}
SPL {X  -160.000, Y  +400.690, Z    +0.000, E1   +14.484, E3 +119347.603}
SPL {X  -160.000, Y  +398.391, Z    +0.000, E1   +14.502, E3 +119366.429}
SPL {X  -160.000, Y  +395.999, Z    +0.000, E1   +14.484, E3 +119386.219}
SPL {X  -160.000, Y  +393.685, Z    +0.000, E1   +14.486, E3 +119405.291}
SPL {X  -159.999, Y  +391.313, Z    +0.000, E1   +14.479, E3 +119424.873}
SPL {X  -159.970, Y  +388.900, Z    +0.000, E1   +14.480, E3 +119444.757}
SPL {X  -159.903, Y  +386.417, Z    +0.000, E1   +14.475, E3 +119465.263}
SPL {X  -159.796, Y  +383.921, Z    +0.000, E1   +14.466, E3 +119485.918}
SPL {X  -159.651, Y  +381.443, Z    +0.000, E1   +14.453, E3 +119506.466}
SPL {X  -159.474, Y  +379.042, Z    +0.000, E1   +14.434, E3 +119526.430}
SPL {X  -159.316, Y  +377.219, Z    +0.000, E1   +14.400, E3 +119541.658}
ENDSPLINE

SPLINE
SPL {X  -159.452, Y  +378.767, Z    +0.000, E1   +11.887, E3 +119562.647}
SPL {X  -159.840, Y  +384.856, Z    +0.000, E1    +7.126, E3 +119581.619}
SPL {X  -159.991, Y  +390.336, Z    +0.000, E1    +2.803, E3 +119595.442}
SPL {X  -160.000, Y  +403.532, Z    +0.000, E1    -6.523, E3 +119613.162}
SPL {X  -160.000, Y  +409.023, Z    +0.000, E1   -10.003, E3 +119623.936}
SPL {X  -160.000, Y  +418.032, Z    +0.000, E1   -14.569, E3 +119648.795}
SPL {X  -160.000, Y  +420.561, Z    +0.000, E1   -14.816, E3 +119666.275}
SPL {X  -160.000, Y  +422.801, Z    +0.000, E1   -14.823, E3 +119684.224}
SPL {X  -160.000, Y  +425.518, Z    +0.000, E1   -14.845, E3 +119705.998}
SPL {X  -160.000, Y  +428.688, Z    +0.000, E1   -14.854, E3 +119731.407}
SPL {X  -160.000, Y  +431.971, Z    +0.000, E1   -14.849, E3 +119757.875}
SPL {X  -160.000, Y  +435.345, Z    +0.000, E1   -14.857, E3 +119784.925}
SPL {X  -160.000, Y  +438.732, Z    +0.000, E1   -14.858, E3 +119812.074}
SPL {X  -160.000, Y  +441.925, Z    +0.000, E1   -14.848, E3 +119837.744}
SPL {X  -160.000, Y  +444.299, Z    +0.000, E1   -14.809, E3 +119856.929}
SPL {X  -160.000, Y  +446.229, Z    +0.000, E1   -14.820, E3 +119872.348}
SPL {X  -160.000, Y  +448.987, Z    +0.000, E1   -14.868, E3 +119894.284}
SPL {X  -160.000, Y  +452.351, Z    +0.000, E1   -14.871, E3 +119921.260}
SPL {X  -160.000, Y  +455.709, Z    +0.000, E1   -14.880, E3 +119948.075}
SPL {X  -160.000, Y  +458.189, Z    +0.000, E1   -14.832, E3 +119968.076}
SPL {X  -160.000, Y  +459.885, Z    +0.000, E1   -14.825, E3 +119981.747}
SPL {X  -160.000, Y  +462.438, Z    +0.000, E1   -14.868, E3 +120002.157}
SPL {X  -160.000, Y  +465.575, Z    +0.000, E1   -14.849, E3 +120027.465}
SPL {X  -160.000, Y  +468.581, Z    +0.000, E1   -14.841, E3 +120051.697}
SPL {X  -160.000, Y  +471.795, Z    +0.000, E1   -14.854, E3 +120077.485}
SPL {X  -160.000, Y  +475.138, Z    +0.000, E1   -14.853, E3 +120104.335}
SPL {X  -160.000, Y  +477.981, Z    +0.000, E1   -14.823, E3 +120127.256}
SPL {X  -160.000, Y  +480.658, Z    +0.000, E1   -14.835, E3 +120148.732}
SPL {X  -160.000, Y  +483.534, Z    +0.000, E1   -14.838, E3 +120171.826}
SPL {X  -160.000, Y  +486.226, Z    +0.000, E1   -14.823, E3 +120193.491}
SPL {X  -160.000, Y  +488.751, Z    +0.000, E1   -14.827, E3 +120213.764}
SPL {X  -160.000, Y  +491.612, Z    +0.000, E1   -14.844, E3 +120236.687}
SPL {X  -160.000, Y  +494.417, Z    +0.000, E1   -14.827, E3 +120259.277}
SPL {X  -160.000, Y  +496.961, Z    +0.000, E1   -14.824, E3 +120279.721}
SPL {X  -160.000, Y  +499.610, Z    +0.000, E1   -14.830, E3 +120300.994}
SPL {X  -160.000, Y  +502.268, Z    +0.000, E1   -14.832, E3 +120322.263}
SPL {X  -160.000, Y  +505.041, Z    +0.000, E1   -14.849, E3 +120344.426}
SPL {X  -160.000, Y  +507.743, Z    +0.000, E1   -14.842, E3 +120366.050}
SPL {X  -160.000, Y  +510.437, Z    +0.000, E1   -14.860, E3 +120387.563}
SPL {X  -160.000, Y  +513.179, Z    +0.000, E1   -14.849, E3 +120409.611}
SPL {X  -160.000, Y  +515.613, Z    +0.000, E1   -14.829, E3 +120429.281}
SPL {X  -160.000, Y  +518.188, Z    +0.000, E1   -14.845, E3 +120449.911}
SPL {X  -160.000, Y  +520.790, Z    +0.000, E1   -14.839, E3 +120470.739}
SPL {X  -160.000, Y  +523.469, Z    +0.000, E1   -14.855, E3 +120492.188}
SPL {X  -160.000, Y  +526.403, Z    +0.000, E1   -14.858, E3 +120515.724}
SPL {X  -160.000, Y  +529.266, Z    +0.000, E1   -14.848, E3 +120538.731}
SPL {X  -160.000, Y  +531.688, Z    +0.000, E1   -14.826, E3 +120558.281}
SPL {X  -160.000, Y  +534.214, Z    +0.000, E1   -14.841, E3 +120578.544}
SPL {X  -160.000, Y  +537.002, Z    +0.000, E1   -14.839, E3 +120600.962}
SPL {X  -160.000, Y  +539.729, Z    +0.000, E1   -14.840, E3 +120622.774}
SPL {X  -160.000, Y  +542.408, Z    +0.000, E1   -14.839, E3 +120644.327}
SPL {X  -160.000, Y  +545.014, Z    +0.000, E1   -14.831, E3 +120665.272}
SPL {X  -160.000, Y  +547.659, Z    +0.000, E1   -14.839, E3 +120686.487}
SPL {X  -160.000, Y  +550.215, Z    +0.000, E1   -14.827, E3 +120707.052}
SPL {X  -160.000, Y  +552.762, Z    +0.000, E1   -14.836, E3 +120727.470}
SPL {X  -160.000, Y  +555.331, Z    +0.000, E1   -14.837, E3 +120748.011}
SPL {X  -160.000, Y  +558.235, Z    +0.000, E1   -14.869, E3 +120771.174}
SPL {X  -160.000, Y  +561.088, Z    +0.000, E1   -14.848, E3 +120794.093}
SPL {X  -160.000, Y  +563.693, Z    +0.000, E1   -14.852, E3 +120814.953}
SPL {X  -160.000, Y  +566.560, Z    +0.000, E1   -14.865, E3 +120837.931}
SPL {X  -160.000, Y  +569.305, Z    +0.000, E1   -14.848, E3 +120859.959}
SPL {X  -160.000, Y  +571.769, Z    +0.000, E1   -14.852, E3 +120879.705}
SPL {X  -160.000, Y  +574.366, Z    +0.000, E1   -14.855, E3 +120900.492}
SPL {X  -160.000, Y  +577.037, Z    +0.000, E1   -14.859, E3 +120921.892}
SPL {X  -160.000, Y  +579.855, Z    +0.000, E1   -14.869, E3 +120944.419}
SPL {X  -160.000, Y  +582.456, Z    +0.000, E1   -14.854, E3 +120965.279}
SPL {X  -160.000, Y  +585.083, Z    +0.000, E1   -14.866, E3 +120986.329}
SPL {X  -160.000, Y  +587.675, Z    +0.000, E1   -14.853, E3 +121007.120}
SPL {X  -160.000, Y  +590.216, Z    +0.000, E1   -14.864, E3 +121027.439}
SPL {X  -160.000, Y  +592.848, Z    +0.000, E1   -14.865, E3 +121048.490}
SPL {X  -160.000, Y  +595.342, Z    +0.000, E1   -14.848, E3 +121068.668}
SPL {X  -160.000, Y  +597.995, Z    +0.000, E1   -14.848, E3 +121090.007}
SPL {X  -160.000, Y  +600.731, Z    +0.000, E1   -14.846, E3 +121111.959}
SPL {X  -160.000, Y  +603.404, Z    +0.000, E1   -14.846, E3 +121133.395}
SPL {X  -160.000, Y  +605.923, Z    +0.000, E1   -14.838, E3 +121153.636}
SPL {X  -160.000, Y  +608.492, Z    +0.000, E1   -14.846, E3 +121174.239}
SPL {X  -160.000, Y  +611.345, Z    +0.000, E1   -14.856, E3 +121197.097}
SPL {X  -160.000, Y  +614.087, Z    +0.000, E1   -14.839, E3 +121219.157}
SPL {X  -160.000, Y  +616.566, Z    +0.000, E1   -14.839, E3 +121239.051}
SPL {X  -160.000, Y  +619.350, Z    +0.000, E1   -14.855, E3 +121261.339}
SPL {X  -160.000, Y  +622.198, Z    +0.000, E1   -14.846, E3 +121284.223}
SPL {X  -160.000, Y  +624.642, Z    +0.000, E1   -14.829, E3 +121303.896}
SPL {X  -160.000, Y  +627.119, Z    +0.000, E1   -14.843, E3 +121323.736}
SPL {X  -160.000, Y  +629.682, Z    +0.000, E1   -14.838, E3 +121344.305}
SPL {X  -160.000, Y  +632.223, Z    +0.000, E1   -14.841, E3 +121364.696}
SPL {X  -160.000, Y  +634.941, Z    +0.000, E1   -14.846, E3 +121386.493}
SPL {X  -160.000, Y  +637.723, Z    +0.000, E1   -14.844, E3 +121408.838}
SPL {X  -160.000, Y  +640.315, Z    +0.000, E1   -14.836, E3 +121429.635}
SPL {X  -160.000, Y  +643.085, Z    +0.000, E1   -14.865, E3 +121451.687}
SPL {X  -160.000, Y  +645.845, Z    +0.000, E1   -14.848, E3 +121473.875}
SPL {X  -160.000, Y  +648.229, Z    +0.000, E1   -14.834, E3 +121493.085}
SPL {X  -160.000, Y  +650.656, Z    +0.000, E1   -14.835, E3 +121512.641}
SPL {X  -160.000, Y  +653.134, Z    +0.000, E1   -14.827, E3 +121532.568}
SPL {X  -160.000, Y  +655.670, Z    +0.000, E1   -14.841, E3 +121552.862}
SPL {X  -160.000, Y  +658.349, Z    +0.000, E1   -14.842, E3 +121574.338}
SPL {X  -160.000, Y  +660.936, Z    +0.000, E1   -14.838, E3 +121595.090}
SPL {X  -160.000, Y  +663.567, Z    +0.000, E1   -14.845, E3 +121616.220}
SPL {X  -160.000, Y  +666.216, Z    +0.000, E1   -14.832, E3 +121637.536}
SPL {X  -159.997, Y  +668.731, Z    +0.000, E1   -14.834, E3 +121657.728}
SPL {X  -159.962, Y  +671.176, Z    +0.000, E1   -14.822, E3 +121677.440}
SPL {X  -159.895, Y  +673.507, Z    +0.000, E1   -14.821, E3 +121696.171}
SPL {X  -159.785, Y  +675.985, Z    +0.000, E1   -14.818, E3 +121716.172}
SPL {X  -159.627, Y  +678.622, Z    +0.000, E1   -14.804, E3 +121737.525}
SPL {X  -159.438, Y  +681.094, Z    +0.000, E1   -14.770, E3 +121757.697}
SPL {X  -159.262, Y  +683.054, Z    +0.000, E1   -14.719, E3 +121773.925}
ENDSPLINE

SPLINE
SPL {X  -159.661, Y  +678.114, Z    +0.000, E1    -9.575, E3 +121803.517}
SPL {X  -159.942, Y  +672.020, Z    +0.000, E1    -4.692, E3 +121822.144}
SPL {X  -160.000, Y  +664.971, Z    +0.000, E1    +0.516, E3 +121841.694}
SPL {X  -160.000, Y  +660.032, Z    +0.000, E1    +3.995, E3 +121853.637}
SPL {X  -160.000, Y  +652.280, Z    +0.000, E1    +8.913, E3 +121872.152}
SPL {X  -160.000, Y  +644.147, Z    +0.000, E1   +13.158, E3 +121895.702}
SPL {X  -160.000, Y  +641.594, Z    +0.000, E1   +13.488, E3 +121914.143}
SPL {X  -160.000, Y  +639.799, Z    +0.000, E1   +13.486, E3 +121930.053}
SPL {X  -160.000, Y  +637.896, Z    +0.000, E1   +13.493, E3 +121946.868}
SPL {X  -160.000, Y  +635.832, Z    +0.000, E1   +13.499, E3 +121965.127}
SPL {X  -160.000, Y  +633.839, Z    +0.000, E1   +13.489, E3 +121982.816}
SPL {X  -160.000, Y  +631.625, Z    +0.000, E1   +13.508, E3 +122002.357}
SPL {X  -160.000, Y  +629.417, Z    +0.000, E1   +13.491, E3 +122021.968}
SPL {X  -160.000, Y  +627.180, Z    +0.000, E1   +13.508, E3 +122041.722}
SPL {X  -160.000, Y  +624.970, Z    +0.000, E1   +13.490, E3 +122061.372}
SPL {X  -160.000, Y  +623.020, Z    +0.000, E1   +13.491, E3 +122078.602}
SPL {X  -160.000, Y  +620.888, Z    +0.000, E1   +13.501, E3 +122097.464}
SPL {X  -160.000, Y  +618.790, Z    +0.000, E1   +13.488, E3 +122116.087}
SPL {X  -160.000, Y  +616.631, Z    +0.000, E1   +13.504, E3 +122135.140}
SPL {X  -160.000, Y  +614.230, Z    +0.000, E1   +13.510, E3 +122156.336}
SPL {X  -160.000, Y  +612.132, Z    +0.000, E1   +13.485, E3 +122175.053}
SPL {X  -160.000, Y  +610.405, Z    +0.000, E1   +13.477, E3 +122190.426}
SPL {X  -160.000, Y  +608.437, Z    +0.000, E1   +13.502, E3 +122207.681}
SPL {X  -160.000, Y  +606.281, Z    +0.000, E1   +13.502, E3 +122226.699}
SPL {X  -160.000, Y  +604.124, Z    +0.000, E1   +13.513, E3 +122245.754}
SPL {X  -160.000, Y  +601.878, Z    +0.000, E1   +13.505, E3 +122265.651}
SPL {X  -160.000, Y  +599.648, Z    +0.000, E1   +13.506, E3 +122285.428}
SPL {X  -160.000, Y  +597.673, Z    +0.000, E1   +13.479, E3 +122303.102}
SPL {X  -160.000, Y  +595.601, Z    +0.000, E1   +13.499, E3 +122321.385}
SPL {X  -160.000, Y  +593.187, Z    +0.000, E1   +13.500, E3 +122342.765}
SPL {X  -160.000, Y  +591.079, Z    +0.000, E1   +13.483, E3 +122361.491}
SPL {X  -160.000, Y  +589.151, Z    +0.000, E1   +13.489, E3 +122378.542}
SPL {X  -160.000, Y  +586.908, Z    +0.000, E1   +13.501, E3 +122398.388}
SPL {X  -160.000, Y  +584.660, Z    +0.000, E1   +13.490, E3 +122418.329}
SPL {X  -160.000, Y  +582.409, Z    +0.000, E1   +13.499, E3 +122438.247}
SPL {X  -160.000, Y  +580.150, Z    +0.000, E1   +13.490, E3 +122458.294}
SPL {X  -160.000, Y  +577.953, Z    +0.000, E1   +13.493, E3 +122477.752}
SPL {X  -160.000, Y  +575.630, Z    +0.000, E1   +13.502, E3 +122498.236}
SPL {X  -160.000, Y  +573.418, Z    +0.000, E1   +13.502, E3 +122517.744}
SPL {X  -160.000, Y  +571.226, Z    +0.000, E1   +13.520, E3 +122536.953}
SPL {X  -160.000, Y  +569.166, Z    +0.000, E1   +13.512, E3 +122555.143}
SPL {X  -160.000, Y  +567.275, Z    +0.000, E1   +13.517, E3 +122571.811}
SPL {X  -160.000, Y  +565.259, Z    +0.000, E1   +13.523, E3 +122589.600}
SPL {X  -160.000, Y  +563.305, Z    +0.000, E1   +13.512, E3 +122606.938}
SPL {X  -160.000, Y  +561.240, Z    +0.000, E1   +13.521, E3 +122625.200}
SPL {X  -160.000, Y  +558.881, Z    +0.000, E1   +13.524, E3 +122646.042}
SPL {X  -160.000, Y  +556.697, Z    +0.000, E1   +13.510, E3 +122665.428}
SPL {X  -160.000, Y  +554.624, Z    +0.000, E1   +13.512, E3 +122683.759}
SPL {X  -160.000, Y  +552.465, Z    +0.000, E1   +13.514, E3 +122702.843}
SPL {X  -160.000, Y  +550.315, Z    +0.000, E1   +13.514, E3 +122721.837}
SPL {X  -160.000, Y  +548.056, Z    +0.000, E1   +13.519, E3 +122741.838}
SPL {X  -160.000, Y  +545.826, Z    +0.000, E1   +13.501, E3 +122761.716}
SPL {X  -160.000, Y  +543.677, Z    +0.000, E1   +13.502, E3 +122780.773}
SPL {X  -160.000, Y  +541.664, Z    +0.000, E1   +13.489, E3 +122798.659}
SPL {X  -160.000, Y  +539.659, Z    +0.000, E1   +13.494, E3 +122816.419}
SPL {X  -160.000, Y  +537.370, Z    +0.000, E1   +13.501, E3 +122836.658}
SPL {X  -160.000, Y  +535.056, Z    +0.000, E1   +13.506, E3 +122857.054}
SPL {X  -160.000, Y  +532.975, Z    +0.000, E1   +13.494, E3 +122875.540}
SPL {X  -160.000, Y  +530.925, Z    +0.000, E1   +13.499, E3 +122893.702}
SPL {X  -160.000, Y  +528.768, Z    +0.000, E1   +13.498, E3 +122912.803}
SPL {X  -160.000, Y  +526.547, Z    +0.000, E1   +13.499, E3 +122932.472}
SPL {X  -160.000, Y  +523.964, Z    +0.000, E1   +13.742, E3 +122951.977}
SPL {X  -160.000, Y  +513.971, Z    +0.000, E1   +18.644, E3 +122970.889}
SPL {X  -160.000, Y  +513.562, Z    +0.000, E1   +16.972, E3 +122990.765}
SPL {X  -160.000, Y  +513.358, Z    +0.000, E1   +15.267, E3 +123011.037}
SPL {X  -160.000, Y  +512.244, Z    +0.000, E1   +14.473, E3 +123029.494}
SPL {X  -160.000, Y  +509.675, Z    +0.000, E1   +14.481, E3 +123050.637}
SPL {X  -160.000, Y  +507.162, Z    +0.000, E1   +14.470, E3 +123071.377}
SPL {X  -160.000, Y  +504.735, Z    +0.000, E1   +14.473, E3 +123091.348}
SPL {X  -160.000, Y  +502.261, Z    +0.000, E1   +14.476, E3 +123111.684}
SPL {X  -160.000, Y  +499.798, Z    +0.000, E1   +14.482, E3 +123131.887}
SPL {X  -160.000, Y  +497.435, Z    +0.000, E1   +14.476, E3 +123151.363}
SPL {X  -160.000, Y  +495.089, Z    +0.000, E1   +14.475, E3 +123170.730}
SPL {X  -160.000, Y  +492.764, Z    +0.000, E1   +14.469, E3 +123189.902}
SPL {X  -160.000, Y  +490.292, Z    +0.000, E1   +14.476, E3 +123210.303}
SPL {X  -160.000, Y  +487.641, Z    +0.000, E1   +14.470, E3 +123232.199}
SPL {X  -160.000, Y  +485.054, Z    +0.000, E1   +14.460, E3 +123253.641}
SPL {X  -160.000, Y  +482.421, Z    +0.000, E1   +14.461, E3 +123275.360}
SPL {X  -160.000, Y  +480.000, Z    +0.000, E1   +14.451, E3 +123295.324}
SPL {X  -160.000, Y  +477.551, Z    +0.000, E1   +14.466, E3 +123315.452}
SPL {X  -160.000, Y  +475.253, Z    +0.000, E1   +14.450, E3 +123334.427}
SPL {X  -160.000, Y  +473.070, Z    +0.000, E1   +14.454, E3 +123352.448}
SPL {X  -160.000, Y  +470.603, Z    +0.000, E1   +14.464, E3 +123372.748}
SPL {X  -160.000, Y  +468.243, Z    +0.000, E1   +14.458, E3 +123392.147}
SPL {X  -160.000, Y  +465.791, Z    +0.000, E1   +14.475, E3 +123412.291}
SPL {X  -160.000, Y  +463.103, Z    +0.000, E1   +14.474, E3 +123434.440}
SPL {X  -160.000, Y  +460.743, Z    +0.000, E1   +14.465, E3 +123453.848}
SPL {X  -160.000, Y  +458.292, Z    +0.000, E1   +14.492, E3 +123473.847}
SPL {X  -160.000, Y  +455.874, Z    +0.000, E1   +14.484, E3 +123493.705}
SPL {X  -160.000, Y  +453.555, Z    +0.000, E1   +14.488, E3 +123512.784}
SPL {X  -160.000, Y  +451.093, Z    +0.000, E1   +14.485, E3 +123533.096}
SPL {X  -160.000, Y  +448.700, Z    +0.000, E1   +14.483, E3 +123552.786}
SPL {X  -160.000, Y  +446.277, Z    +0.000, E1   +14.485, E3 +123572.709}
SPL {X  -160.000, Y  +443.879, Z    +0.000, E1   +14.485, E3 +123592.448}
SPL {X  -160.000, Y  +441.447, Z    +0.000, E1   +14.485, E3 +123612.455}
SPL {X  -160.000, Y  +439.006, Z    +0.000, E1   +14.488, E3 +123632.538}
SPL {X  -160.000, Y  +436.311, Z    +0.000, E1   +14.498, E3 +123654.697}
SPL {X  -160.000, Y  +433.559, Z    +0.000, E1   +14.491, E3 +123677.366}
SPL {X  -160.000, Y  +431.162, Z    +0.000, E1   +14.479, E3 +123697.117}
SPL {X  -160.000, Y  +429.152, Z    +0.000, E1   +14.469, E3 +123713.699}
SPL {X  -160.000, Y  +426.863, Z    +0.000, E1   +14.490, E3 +123732.478}
SPL {X  -160.000, Y  +424.653, Z    +0.000, E1   +14.467, E3 +123750.737}
SPL {X  -160.000, Y  +422.337, Z    +0.000, E1   +14.492, E3 +123769.721}
SPL {X  -160.000, Y  +419.639, Z    +0.000, E1   +14.504, E3 +123791.761}
SPL {X  -160.000, Y  +417.127, Z    +0.000, E1   +14.501, E3 +123812.353}
SPL {X  -160.000, Y  +414.849, Z    +0.000, E1   +14.496, E3 +123831.087}
SPL {X  -160.000, Y  +412.396, Z    +0.000, E1   +14.505, E3 +123851.276}
SPL {X  -160.000, Y  +409.815, Z    +0.000, E1   +14.498, E3 +123872.530}
SPL {X  -160.000, Y  +407.614, Z    +0.000, E1   +14.484, E3 +123890.655}
SPL {X  -160.000, Y  +405.406, Z    +0.000, E1   +14.501, E3 +123908.718}
SPL {X  -160.000, Y  +402.958, Z    +0.000, E1   +14.500, E3 +123928.888}
SPL {X  -160.000, Y  +400.690, Z    +0.000, E1   +14.484, E3 +123947.600}
SPL {X  -160.000, Y  +398.391, Z    +0.000, E1   +14.502, E3 +123966.426}
SPL {X  -160.000, Y  +395.999, Z    +0.000, E1   +14.484, E3 +123986.216}
SPL {X  -160.000, Y  +393.685, Z    +0.000, E1   +14.486, E3 +124005.288}
SPL {X  -159.999, Y  +391.313, Z    +0.000, E1   +14.479, E3 +124024.870}
SPL {X  -159.970, Y  +388.900, Z    +0.000, E1   +14.480, E3 +124044.754}
SPL {X  -159.903, Y  +386.417, Z    +0.000, E1   +14.475, E3 +124065.259}
SPL {X  -159.796, Y  +383.921, Z    +0.000, E1   +14.466, E3 +124085.915}
SPL {X  -159.651, Y  +381.443, Z    +0.000, E1   +14.453, E3 +124106.463}
SPL {X  -159.474, Y  +379.042, Z    +0.000, E1   +14.434, E3 +124126.427}
SPL {X  -159.316, Y  +377.219, Z    +0.000, E1   +14.400, E3 +124141.655}
ENDSPLINE

SPLINE
SPL {X  -159.452, Y  +378.767, Z    +0.000, E1   +11.887, E3 +124162.644}
SPL {X  -159.840, Y  +384.856, Z    +0.000, E1    +7.126, E3 +124181.616}
SPL {X  -159.991, Y  +390.336, Z    +0.000, E1    +2.803, E3 +124195.439}
SPL {X  -160.000, Y  +403.532, Z    +0.000, E1    -6.523, E3 +124213.159}
SPL {X  -160.000, Y  +409.023, Z    +0.000, E1   -10.003, E3 +124223.933}
SPL {X  -160.000, Y  +418.032, Z    +0.000, E1   -14.569, E3 +124248.792}
SPL {X  -160.000, Y  +420.561, Z    +0.000, E1   -14.816, E3 +124266.272}
SPL {X  -160.000, Y  +422.801, Z    +0.000, E1   -14.823, E3 +124284.221}
SPL {X  -160.000, Y  +425.518, Z    +0.000, E1   -14.845, E3 +124305.995}
SPL {X  -160.000, Y  +428.688, Z    +0.000, E1   -14.854, E3 +124331.403}
SPL {X  -160.000, Y  +431.971, Z    +0.000, E1   -14.849, E3 +124357.872}
SPL {X  -160.000, Y  +435.345, Z    +0.000, E1   -14.857, E3 +124384.922}
SPL {X  -160.000, Y  +438.732, Z    +0.000, E1   -14.858, E3 +124412.071}
SPL {X  -160.000, Y  +441.925, Z    +0.000, E1   -14.848, E3 +124437.741}
SPL {X  -160.000, Y  +444.299, Z    +0.000, E1   -14.809, E3 +124456.926}
SPL {X  -160.000, Y  +446.229, Z    +0.000, E1   -14.820, E3 +124472.345}
SPL {X  -160.000, Y  +448.987, Z    +0.000, E1   -14.868, E3 +124494.281}
SPL {X  -160.000, Y  +452.351, Z    +0.000, E1   -14.871, E3 +124521.257}
SPL {X  -160.000, Y  +455.709, Z    +0.000, E1   -14.880, E3 +124548.071}
SPL {X  -160.000, Y  +458.189, Z    +0.000, E1   -14.832, E3 +124568.073}
SPL {X  -160.000, Y  +459.885, Z    +0.000, E1   -14.825, E3 +124581.744}
SPL {X  -160.000, Y  +462.438, Z    +0.000, E1   -14.868, E3 +124602.154}
SPL {X  -160.000, Y  +465.575, Z    +0.000, E1   -14.849, E3 +124627.462}
SPL {X  -160.000, Y  +468.581, Z    +0.000, E1   -14.841, E3 +124651.694}
SPL {X  -160.000, Y  +471.795, Z    +0.000, E1   -14.854, E3 +124677.482}
SPL {X  -160.000, Y  +475.138, Z    +0.000, E1   -14.853, E3 +124704.332}
SPL {X  -160.000, Y  +477.981, Z    +0.000, E1   -14.823, E3 +124727.252}
SPL {X  -160.000, Y  +480.658, Z    +0.000, E1   -14.835, E3 +124748.728}
SPL {X  -160.000, Y  +483.534, Z    +0.000, E1   -14.838, E3 +124771.823}
SPL {X  -160.000, Y  +486.226, Z    +0.000, E1   -14.823, E3 +124793.488}
SPL {X  -160.000, Y  +488.751, Z    +0.000, E1   -14.827, E3 +124813.761}
SPL {X  -160.000, Y  +491.612, Z    +0.000, E1   -14.844, E3 +124836.683}
SPL {X  -160.000, Y  +494.417, Z    +0.000, E1   -14.827, E3 +124859.274}
SPL {X  -160.000, Y  +496.961, Z    +0.000, E1   -14.824, E3 +124879.718}
SPL {X  -160.000, Y  +499.610, Z    +0.000, E1   -14.830, E3 +124900.991}
SPL {X  -160.000, Y  +502.268, Z    +0.000, E1   -14.832, E3 +124922.260}
SPL {X  -160.000, Y  +505.041, Z    +0.000, E1   -14.849, E3 +124944.423}
SPL {X  -160.000, Y  +507.743, Z    +0.000, E1   -14.842, E3 +124966.046}
SPL {X  -160.000, Y  +510.437, Z    +0.000, E1   -14.860, E3 +124987.560}
SPL {X  -160.000, Y  +513.179, Z    +0.000, E1   -14.849, E3 +125009.608}
SPL {X  -160.000, Y  +515.613, Z    +0.000, E1   -14.829, E3 +125029.278}
SPL {X  -160.000, Y  +518.188, Z    +0.000, E1   -14.845, E3 +125049.907}
SPL {X  -160.000, Y  +520.790, Z    +0.000, E1   -14.839, E3 +125070.736}
SPL {X  -160.000, Y  +523.469, Z    +0.000, E1   -14.855, E3 +125092.184}
SPL {X  -160.000, Y  +526.403, Z    +0.000, E1   -14.858, E3 +125115.721}
SPL {X  -160.000, Y  +529.266, Z    +0.000, E1   -14.848, E3 +125138.728}
SPL {X  -160.000, Y  +531.688, Z    +0.000, E1   -14.826, E3 +125158.278}
SPL {X  -160.000, Y  +534.214, Z    +0.000, E1   -14.841, E3 +125178.541}
SPL {X  -160.000, Y  +537.002, Z    +0.000, E1   -14.839, E3 +125200.959}
SPL {X  -160.000, Y  +539.729, Z    +0.000, E1   -14.840, E3 +125222.771}
SPL {X  -160.000, Y  +542.408, Z    +0.000, E1   -14.839, E3 +125244.324}
SPL {X  -160.000, Y  +545.014, Z    +0.000, E1   -14.831, E3 +125265.269}
SPL {X  -160.000, Y  +547.659, Z    +0.000, E1   -14.839, E3 +125286.483}
SPL {X  -160.000, Y  +550.215, Z    +0.000, E1   -14.827, E3 +125307.048}
SPL {X  -160.000, Y  +552.762, Z    +0.000, E1   -14.836, E3 +125327.467}
SPL {X  -160.000, Y  +555.331, Z    +0.000, E1   -14.837, E3 +125348.008}
SPL {X  -160.000, Y  +558.235, Z    +0.000, E1   -14.869, E3 +125371.171}
SPL {X  -160.000, Y  +561.088, Z    +0.000, E1   -14.848, E3 +125394.090}
SPL {X  -160.000, Y  +563.693, Z    +0.000, E1   -14.852, E3 +125414.950}
SPL {X  -160.000, Y  +566.560, Z    +0.000, E1   -14.865, E3 +125437.928}
SPL {X  -160.000, Y  +569.305, Z    +0.000, E1   -14.848, E3 +125459.956}
SPL {X  -160.000, Y  +571.769, Z    +0.000, E1   -14.852, E3 +125479.702}
SPL {X  -160.000, Y  +574.366, Z    +0.000, E1   -14.855, E3 +125500.489}
SPL {X  -160.000, Y  +577.037, Z    +0.000, E1   -14.859, E3 +125521.889}
SPL {X  -160.000, Y  +579.855, Z    +0.000, E1   -14.869, E3 +125544.416}
SPL {X  -160.000, Y  +582.456, Z    +0.000, E1   -14.854, E3 +125565.276}
SPL {X  -160.000, Y  +585.083, Z    +0.000, E1   -14.866, E3 +125586.325}
SPL {X  -160.000, Y  +587.675, Z    +0.000, E1   -14.853, E3 +125607.116}
SPL {X  -160.000, Y  +590.216, Z    +0.000, E1   -14.864, E3 +125627.436}
SPL {X  -160.000, Y  +592.848, Z    +0.000, E1   -14.865, E3 +125648.487}
SPL {X  -160.000, Y  +595.342, Z    +0.000, E1   -14.848, E3 +125668.664}
SPL {X  -160.000, Y  +597.995, Z    +0.000, E1   -14.848, E3 +125690.004}
SPL {X  -160.000, Y  +600.731, Z    +0.000, E1   -14.846, E3 +125711.956}
SPL {X  -160.000, Y  +603.404, Z    +0.000, E1   -14.846, E3 +125733.392}
SPL {X  -160.000, Y  +605.923, Z    +0.000, E1   -14.838, E3 +125753.632}
SPL {X  -160.000, Y  +608.492, Z    +0.000, E1   -14.846, E3 +125774.236}
SPL {X  -160.000, Y  +611.345, Z    +0.000, E1   -14.856, E3 +125797.094}
SPL {X  -160.000, Y  +614.087, Z    +0.000, E1   -14.839, E3 +125819.154}
SPL {X  -160.000, Y  +616.566, Z    +0.000, E1   -14.839, E3 +125839.047}
SPL {X  -160.000, Y  +619.350, Z    +0.000, E1   -14.855, E3 +125861.335}
SPL {X  -160.000, Y  +622.198, Z    +0.000, E1   -14.846, E3 +125884.220}
SPL {X  -160.000, Y  +624.642, Z    +0.000, E1   -14.829, E3 +125903.893}
SPL {X  -160.000, Y  +627.119, Z    +0.000, E1   -14.843, E3 +125923.732}
SPL {X  -160.000, Y  +629.682, Z    +0.000, E1   -14.838, E3 +125944.301}
SPL {X  -160.000, Y  +632.223, Z    +0.000, E1   -14.841, E3 +125964.693}
SPL {X  -160.000, Y  +634.941, Z    +0.000, E1   -14.846, E3 +125986.490}
SPL {X  -160.000, Y  +637.723, Z    +0.000, E1   -14.844, E3 +126008.834}
SPL {X  -160.000, Y  +640.315, Z    +0.000, E1   -14.836, E3 +126029.632}
SPL {X  -160.000, Y  +643.085, Z    +0.000, E1   -14.865, E3 +126051.684}
SPL {X  -160.000, Y  +645.845, Z    +0.000, E1   -14.848, E3 +126073.872}
SPL {X  -160.000, Y  +648.229, Z    +0.000, E1   -14.834, E3 +126093.081}
SPL {X  -160.000, Y  +650.656, Z    +0.000, E1   -14.835, E3 +126112.638}
SPL {X  -160.000, Y  +653.134, Z    +0.000, E1   -14.827, E3 +126132.565}
SPL {X  -160.000, Y  +655.670, Z    +0.000, E1   -14.841, E3 +126152.859}
SPL {X  -160.000, Y  +658.349, Z    +0.000, E1   -14.842, E3 +126174.335}
SPL {X  -160.000, Y  +660.936, Z    +0.000, E1   -14.838, E3 +126195.086}
SPL {X  -160.000, Y  +663.567, Z    +0.000, E1   -14.845, E3 +126216.217}
SPL {X  -160.000, Y  +666.216, Z    +0.000, E1   -14.832, E3 +126237.533}
SPL {X  -159.997, Y  +668.731, Z    +0.000, E1   -14.834, E3 +126257.725}
SPL {X  -159.962, Y  +671.176, Z    +0.000, E1   -14.822, E3 +126277.436}
SPL {X  -159.895, Y  +673.507, Z    +0.000, E1   -14.821, E3 +126296.168}
SPL {X  -159.785, Y  +675.985, Z    +0.000, E1   -14.818, E3 +126316.169}
SPL {X  -159.627, Y  +678.622, Z    +0.000, E1   -14.804, E3 +126337.522}
SPL {X  -159.438, Y  +681.094, Z    +0.000, E1   -14.770, E3 +126357.693}
SPL {X  -159.262, Y  +683.054, Z    +0.000, E1   -14.719, E3 +126373.922}
ENDSPLINE

SPLINE
SPL {X  -159.661, Y  +678.114, Z    +0.000, E1    -9.575, E3 +126403.514}
SPL {X  -159.942, Y  +672.020, Z    +0.000, E1    -4.692, E3 +126422.141}
SPL {X  -160.000, Y  +664.971, Z    +0.000, E1    +0.516, E3 +126441.691}
SPL {X  -160.000, Y  +660.032, Z    +0.000, E1    +3.995, E3 +126453.634}
SPL {X  -160.000, Y  +652.280, Z    +0.000, E1    +8.913, E3 +126472.149}
SPL {X  -160.000, Y  +644.147, Z    +0.000, E1   +13.158, E3 +126495.699}
SPL {X  -160.000, Y  +641.594, Z    +0.000, E1   +13.488, E3 +126514.140}
SPL {X  -160.000, Y  +639.799, Z    +0.000, E1   +13.486, E3 +126530.050}
SPL {X  -160.000, Y  +637.896, Z    +0.000, E1   +13.493, E3 +126546.865}
SPL {X  -160.000, Y  +635.832, Z    +0.000, E1   +13.499, E3 +126565.124}
SPL {X  -160.000, Y  +633.839, Z    +0.000, E1   +13.489, E3 +126582.813}
SPL {X  -160.000, Y  +631.625, Z    +0.000, E1   +13.508, E3 +126602.354}
SPL {X  -160.000, Y  +629.417, Z    +0.000, E1   +13.491, E3 +126621.965}
SPL {X  -160.000, Y  +627.180, Z    +0.000, E1   +13.508, E3 +126641.719}
SPL {X  -160.000, Y  +624.970, Z    +0.000, E1   +13.490, E3 +126661.369}
SPL {X  -160.000, Y  +623.020, Z    +0.000, E1   +13.491, E3 +126678.599}
SPL {X  -160.000, Y  +620.888, Z    +0.000, E1   +13.501, E3 +126697.461}
SPL {X  -160.000, Y  +618.790, Z    +0.000, E1   +13.488, E3 +126716.084}
SPL {X  -160.000, Y  +616.631, Z    +0.000, E1   +13.504, E3 +126735.137}
SPL {X  -160.000, Y  +614.230, Z    +0.000, E1   +13.510, E3 +126756.333}
SPL {X  -160.000, Y  +612.132, Z    +0.000, E1   +13.485, E3 +126775.049}
SPL {X  -160.000, Y  +610.405, Z    +0.000, E1   +13.477, E3 +126790.423}
SPL {X  -160.000, Y  +608.437, Z    +0.000, E1   +13.502, E3 +126807.678}
SPL {X  -160.000, Y  +606.281, Z    +0.000, E1   +13.502, E3 +126826.696}
SPL {X  -160.000, Y  +604.124, Z    +0.000, E1   +13.513, E3 +126845.751}
SPL {X  -160.000, Y  +601.878, Z    +0.000, E1   +13.505, E3 +126865.648}
SPL {X  -160.000, Y  +599.648, Z    +0.000, E1   +13.506, E3 +126885.425}
SPL {X  -160.000, Y  +597.673, Z    +0.000, E1   +13.479, E3 +126903.099}
SPL {X  -160.000, Y  +595.601, Z    +0.000, E1   +13.499, E3 +126921.382}
SPL {X  -160.000, Y  +593.187, Z    +0.000, E1   +13.500, E3 +126942.762}
SPL {X  -160.000, Y  +591.079, Z    +0.000, E1   +13.483, E3 +126961.488}
SPL {X  -160.000, Y  +589.151, Z    +0.000, E1   +13.489, E3 +126978.539}
SPL {X  -160.000, Y  +586.908, Z    +0.000, E1   +13.501, E3 +126998.384}
SPL {X  -160.000, Y  +584.660, Z    +0.000, E1   +13.490, E3 +127018.326}
SPL {X  -160.000, Y  +582.409, Z    +0.000, E1   +13.499, E3 +127038.244}
SPL {X  -160.000, Y  +580.150, Z    +0.000, E1   +13.490, E3 +127058.291}
SPL {X  -160.000, Y  +577.953, Z    +0.000, E1   +13.493, E3 +127077.749}
SPL {X  -160.000, Y  +575.630, Z    +0.000, E1   +13.502, E3 +127098.233}
SPL {X  -160.000, Y  +573.418, Z    +0.000, E1   +13.502, E3 +127117.741}
SPL {X  -160.000, Y  +571.226, Z    +0.000, E1   +13.520, E3 +127136.950}
SPL {X  -160.000, Y  +569.166, Z    +0.000, E1   +13.512, E3 +127155.140}
SPL {X  -160.000, Y  +567.275, Z    +0.000, E1   +13.517, E3 +127171.807}
SPL {X  -160.000, Y  +565.259, Z    +0.000, E1   +13.523, E3 +127189.597}
SPL {X  -160.000, Y  +563.305, Z    +0.000, E1   +13.512, E3 +127206.935}
SPL {X  -160.000, Y  +561.240, Z    +0.000, E1   +13.521, E3 +127225.196}
SPL {X  -160.000, Y  +558.881, Z    +0.000, E1   +13.524, E3 +127246.039}
SPL {X  -160.000, Y  +556.697, Z    +0.000, E1   +13.510, E3 +127265.425}
SPL {X  -160.000, Y  +554.624, Z    +0.000, E1   +13.512, E3 +127283.756}
SPL {X  -160.000, Y  +552.465, Z    +0.000, E1   +13.514, E3 +127302.840}
SPL {X  -160.000, Y  +550.315, Z    +0.000, E1   +13.514, E3 +127321.834}
SPL {X  -160.000, Y  +548.056, Z    +0.000, E1   +13.519, E3 +127341.835}
SPL {X  -160.000, Y  +545.826, Z    +0.000, E1   +13.501, E3 +127361.712}
SPL {X  -160.000, Y  +543.677, Z    +0.000, E1   +13.502, E3 +127380.770}
SPL {X  -160.000, Y  +541.664, Z    +0.000, E1   +13.489, E3 +127398.656}
SPL {X  -160.000, Y  +539.659, Z    +0.000, E1   +13.494, E3 +127416.416}
SPL {X  -160.000, Y  +537.370, Z    +0.000, E1   +13.501, E3 +127436.655}
SPL {X  -160.000, Y  +535.056, Z    +0.000, E1   +13.506, E3 +127457.050}
SPL {X  -160.000, Y  +532.975, Z    +0.000, E1   +13.494, E3 +127475.537}
SPL {X  -160.000, Y  +530.925, Z    +0.000, E1   +13.499, E3 +127493.699}
SPL {X  -160.000, Y  +528.768, Z    +0.000, E1   +13.498, E3 +127512.800}
SPL {X  -160.000, Y  +526.547, Z    +0.000, E1   +13.499, E3 +127532.469}
SPL {X  -160.000, Y  +523.964, Z    +0.000, E1   +13.742, E3 +127551.973}
SPL {X  -160.000, Y  +513.971, Z    +0.000, E1   +18.644, E3 +127570.885}
SPL {X  -160.000, Y  +513.562, Z    +0.000, E1   +16.972, E3 +127590.762}
SPL {X  -160.000, Y  +513.358, Z    +0.000, E1   +15.267, E3 +127611.034}
SPL {X  -160.000, Y  +512.244, Z    +0.000, E1   +14.473, E3 +127629.490}
SPL {X  -160.000, Y  +509.675, Z    +0.000, E1   +14.481, E3 +127650.634}
SPL {X  -160.000, Y  +507.162, Z    +0.000, E1   +14.470, E3 +127671.374}
SPL {X  -160.000, Y  +504.735, Z    +0.000, E1   +14.473, E3 +127691.345}
SPL {X  -160.000, Y  +502.261, Z    +0.000, E1   +14.476, E3 +127711.681}
SPL {X  -160.000, Y  +499.798, Z    +0.000, E1   +14.482, E3 +127731.884}
SPL {X  -160.000, Y  +497.435, Z    +0.000, E1   +14.476, E3 +127751.360}
SPL {X  -160.000, Y  +495.089, Z    +0.000, E1   +14.475, E3 +127770.727}
SPL {X  -160.000, Y  +492.764, Z    +0.000, E1   +14.469, E3 +127789.899}
SPL {X  -160.000, Y  +490.292, Z    +0.000, E1   +14.476, E3 +127810.299}
SPL {X  -160.000, Y  +487.641, Z    +0.000, E1   +14.470, E3 +127832.196}
SPL {X  -160.000, Y  +485.054, Z    +0.000, E1   +14.460, E3 +127853.638}
SPL {X  -160.000, Y  +482.421, Z    +0.000, E1   +14.461, E3 +127875.357}
SPL {X  -160.000, Y  +480.000, Z    +0.000, E1   +14.451, E3 +127895.321}
SPL {X  -160.000, Y  +477.551, Z    +0.000, E1   +14.466, E3 +127915.449}
SPL {X  -160.000, Y  +475.253, Z    +0.000, E1   +14.450, E3 +127934.423}
SPL {X  -160.000, Y  +473.070, Z    +0.000, E1   +14.454, E3 +127952.444}
SPL {X  -160.000, Y  +470.603, Z    +0.000, E1   +14.464, E3 +127972.744}
SPL {X  -160.000, Y  +468.243, Z    +0.000, E1   +14.458, E3 +127992.144}
SPL {X  -160.000, Y  +465.791, Z    +0.000, E1   +14.475, E3 +128012.288}
SPL {X  -160.000, Y  +463.103, Z    +0.000, E1   +14.474, E3 +128034.437}
SPL {X  -160.000, Y  +460.743, Z    +0.000, E1   +14.465, E3 +128053.845}
SPL {X  -160.000, Y  +458.292, Z    +0.000, E1   +14.492, E3 +128073.844}
SPL {X  -160.000, Y  +455.874, Z    +0.000, E1   +14.484, E3 +128093.702}
SPL {X  -160.000, Y  +453.555, Z    +0.000, E1   +14.488, E3 +128112.781}
SPL {X  -160.000, Y  +451.093, Z    +0.000, E1   +14.485, E3 +128133.093}
SPL {X  -160.000, Y  +448.700, Z    +0.000, E1   +14.483, E3 +128152.783}
SPL {X  -160.000, Y  +446.277, Z    +0.000, E1   +14.485, E3 +128172.706}
SPL {X  -160.000, Y  +443.879, Z    +0.000, E1   +14.485, E3 +128192.444}
SPL {X  -160.000, Y  +441.447, Z    +0.000, E1   +14.485, E3 +128212.452}
SPL {X  -160.000, Y  +439.006, Z    +0.000, E1   +14.488, E3 +128232.535}
SPL {X  -160.000, Y  +436.311, Z    +0.000, E1   +14.498, E3 +128254.694}
SPL {X  -160.000, Y  +433.559, Z    +0.000, E1   +14.491, E3 +128277.363}
SPL {X  -160.000, Y  +431.162, Z    +0.000, E1   +14.479, E3 +128297.114}
SPL {X  -160.000, Y  +429.152, Z    +0.000, E1   +14.469, E3 +128313.696}
SPL {X  -160.000, Y  +426.863, Z    +0.000, E1   +14.490, E3 +128332.475}
SPL {X  -160.000, Y  +424.653, Z    +0.000, E1   +14.467, E3 +128350.734}
SPL {X  -160.000, Y  +422.337, Z    +0.000, E1   +14.492, E3 +128369.718}
SPL {X  -160.000, Y  +419.639, Z    +0.000, E1   +14.504, E3 +128391.758}
SPL {X  -160.000, Y  +417.127, Z    +0.000, E1   +14.501, E3 +128412.349}
SPL {X  -160.000, Y  +414.849, Z    +0.000, E1   +14.496, E3 +128431.083}
SPL {X  -160.000, Y  +412.396, Z    +0.000, E1   +14.505, E3 +128451.272}
SPL {X  -160.000, Y  +409.815, Z    +0.000, E1   +14.498, E3 +128472.527}
SPL {X  -160.000, Y  +407.614, Z    +0.000, E1   +14.484, E3 +128490.652}
SPL {X  -160.000, Y  +405.406, Z    +0.000, E1   +14.501, E3 +128508.715}
SPL {X  -160.000, Y  +402.958, Z    +0.000, E1   +14.500, E3 +128528.885}
SPL {X  -160.000, Y  +400.690, Z    +0.000, E1   +14.484, E3 +128547.597}
SPL {X  -160.000, Y  +398.391, Z    +0.000, E1   +14.502, E3 +128566.423}
SPL {X  -160.000, Y  +395.999, Z    +0.000, E1   +14.484, E3 +128586.212}
SPL {X  -160.000, Y  +393.685, Z    +0.000, E1   +14.486, E3 +128605.285}
SPL {X  -159.999, Y  +391.313, Z    +0.000, E1   +14.479, E3 +128624.867}
SPL {X  -159.970, Y  +388.900, Z    +0.000, E1   +14.480, E3 +128644.751}
SPL {X  -159.903, Y  +386.417, Z    +0.000, E1   +14.475, E3 +128665.256}
SPL {X  -159.796, Y  +383.921, Z    +0.000, E1   +14.466, E3 +128685.912}
SPL {X  -159.651, Y  +381.443, Z    +0.000, E1   +14.453, E3 +128706.459}
SPL {X  -159.474, Y  +379.042, Z    +0.000, E1   +14.434, E3 +128726.423}
SPL {X  -159.316, Y  +377.219, Z    +0.000, E1   +14.400, E3 +128741.652}
ENDSPLINE

SPLINE
SPL {X  -159.452, Y  +378.767, Z    +0.000, E1   +11.887, E3 +128762.641}
SPL {X  -159.840, Y  +384.856, Z    +0.000, E1    +7.126, E3 +128781.613}
SPL {X  -159.991, Y  +390.336, Z    +0.000, E1    +2.803, E3 +128795.435}
SPL {X  -160.000, Y  +403.532, Z    +0.000, E1    -6.523, E3 +128813.156}
SPL {X  -160.000, Y  +409.023, Z    +0.000, E1   -10.003, E3 +128823.930}
SPL {X  -160.000, Y  +418.032, Z    +0.000, E1   -14.569, E3 +128848.789}
SPL {X  -160.000, Y  +420.561, Z    +0.000, E1   -14.816, E3 +128866.269}
SPL {X  -160.000, Y  +422.801, Z    +0.000, E1   -14.823, E3 +128884.217}
SPL {X  -160.000, Y  +425.518, Z    +0.000, E1   -14.845, E3 +128905.992}
SPL {X  -160.000, Y  +428.688, Z    +0.000, E1   -14.854, E3 +128931.400}
SPL {X  -160.000, Y  +431.971, Z    +0.000, E1   -14.849, E3 +128957.869}
SPL {X  -160.000, Y  +435.345, Z    +0.000, E1   -14.857, E3 +128984.919}
SPL {X  -160.000, Y  +438.732, Z    +0.000, E1   -14.858, E3 +129012.067}
SPL {X  -160.000, Y  +441.925, Z    +0.000, E1   -14.848, E3 +129037.738}
SPL {X  -160.000, Y  +444.299, Z    +0.000, E1   -14.809, E3 +129056.922}
SPL {X  -160.000, Y  +446.229, Z    +0.000, E1   -14.820, E3 +129072.341}
SPL {X  -160.000, Y  +448.987, Z    +0.000, E1   -14.868, E3 +129094.278}
SPL {X  -160.000, Y  +452.351, Z    +0.000, E1   -14.871, E3 +129121.254}
SPL {X  -160.000, Y  +455.709, Z    +0.000, E1   -14.880, E3 +129148.068}
SPL {X  -160.000, Y  +458.189, Z    +0.000, E1   -14.832, E3 +129168.070}
SPL {X  -160.000, Y  +459.885, Z    +0.000, E1   -14.825, E3 +129181.741}
SPL {X  -160.000, Y  +462.438, Z    +0.000, E1   -14.868, E3 +129202.151}
SPL {X  -160.000, Y  +465.575, Z    +0.000, E1   -14.849, E3 +129227.459}
SPL {X  -160.000, Y  +468.581, Z    +0.000, E1   -14.841, E3 +129251.691}
SPL {X  -160.000, Y  +471.795, Z    +0.000, E1   -14.854, E3 +129277.479}
SPL {X  -160.000, Y  +475.138, Z    +0.000, E1   -14.853, E3 +129304.329}
SPL {X  -160.000, Y  +477.981, Z    +0.000, E1   -14.823, E3 +129327.249}
SPL {X  -160.000, Y  +480.658, Z    +0.000, E1   -14.835, E3 +129348.725}
SPL {X  -160.000, Y  +483.534, Z    +0.000, E1   -14.838, E3 +129371.820}
SPL {X  -160.000, Y  +486.226, Z    +0.000, E1   -14.823, E3 +129393.485}
SPL {X  -160.000, Y  +488.751, Z    +0.000, E1   -14.827, E3 +129413.758}
SPL {X  -160.000, Y  +491.612, Z    +0.000, E1   -14.844, E3 +129436.680}
SPL {X  -160.000, Y  +494.417, Z    +0.000, E1   -14.827, E3 +129459.271}
SPL {X  -160.000, Y  +496.961, Z    +0.000, E1   -14.824, E3 +129479.715}
SPL {X  -160.000, Y  +499.610, Z    +0.000, E1   -14.830, E3 +129500.988}
SPL {X  -160.000, Y  +502.268, Z    +0.000, E1   -14.832, E3 +129522.257}
SPL {X  -160.000, Y  +505.041, Z    +0.000, E1   -14.849, E3 +129544.419}
SPL {X  -160.000, Y  +507.743, Z    +0.000, E1   -14.842, E3 +129566.043}
SPL {X  -160.000, Y  +510.437, Z    +0.000, E1   -14.860, E3 +129587.557}
SPL {X  -160.000, Y  +513.179, Z    +0.000, E1   -14.849, E3 +129609.604}
SPL {X  -160.000, Y  +515.613, Z    +0.000, E1   -14.829, E3 +129629.275}
SPL {X  -160.000, Y  +518.188, Z    +0.000, E1   -14.845, E3 +129649.904}
SPL {X  -160.000, Y  +520.790, Z    +0.000, E1   -14.839, E3 +129670.733}
SPL {X  -160.000, Y  +523.469, Z    +0.000, E1   -14.855, E3 +129692.181}
SPL {X  -160.000, Y  +526.403, Z    +0.000, E1   -14.858, E3 +129715.718}
SPL {X  -160.000, Y  +529.266, Z    +0.000, E1   -14.848, E3 +129738.725}
SPL {X  -160.000, Y  +531.688, Z    +0.000, E1   -14.826, E3 +129758.275}
SPL {X  -160.000, Y  +534.214, Z    +0.000, E1   -14.841, E3 +129778.538}
SPL {X  -160.000, Y  +537.002, Z    +0.000, E1   -14.839, E3 +129800.956}
SPL {X  -160.000, Y  +539.729, Z    +0.000, E1   -14.840, E3 +129822.767}
SPL {X  -160.000, Y  +542.408, Z    +0.000, E1   -14.839, E3 +129844.320}
SPL {X  -160.000, Y  +545.014, Z    +0.000, E1   -14.831, E3 +129865.266}
SPL {X  -160.000, Y  +547.659, Z    +0.000, E1   -14.839, E3 +129886.480}
SPL {X  -160.000, Y  +550.215, Z    +0.000, E1   -14.827, E3 +129907.045}
SPL {X  -160.000, Y  +552.762, Z    +0.000, E1   -14.836, E3 +129927.463}
SPL {X  -160.000, Y  +555.331, Z    +0.000, E1   -14.837, E3 +129948.004}
SPL {X  -160.000, Y  +558.235, Z    +0.000, E1   -14.869, E3 +129971.168}
SPL {X  -160.000, Y  +561.088, Z    +0.000, E1   -14.848, E3 +129994.086}
SPL {X  -160.000, Y  +563.693, Z    +0.000, E1   -14.852, E3 +130014.947}
SPL {X  -160.000, Y  +566.560, Z    +0.000, E1   -14.865, E3 +130037.925}
SPL {X  -160.000, Y  +569.305, Z    +0.000, E1   -14.848, E3 +130059.953}
SPL {X  -160.000, Y  +571.769, Z    +0.000, E1   -14.852, E3 +130079.699}
SPL {X  -160.000, Y  +574.366, Z    +0.000, E1   -14.855, E3 +130100.486}
SPL {X  -160.000, Y  +577.037, Z    +0.000, E1   -14.859, E3 +130121.885}
SPL {X  -160.000, Y  +579.855, Z    +0.000, E1   -14.869, E3 +130144.413}
SPL {X  -160.000, Y  +582.456, Z    +0.000, E1   -14.854, E3 +130165.273}
SPL {X  -160.000, Y  +585.083, Z    +0.000, E1   -14.866, E3 +130186.322}
SPL {X  -160.000, Y  +587.675, Z    +0.000, E1   -14.853, E3 +130207.113}
SPL {X  -160.000, Y  +590.216, Z    +0.000, E1   -14.864, E3 +130227.432}
SPL {X  -160.000, Y  +592.848, Z    +0.000, E1   -14.865, E3 +130248.484}
SPL {X  -160.000, Y  +595.342, Z    +0.000, E1   -14.848, E3 +130268.661}
SPL {X  -160.000, Y  +597.995, Z    +0.000, E1   -14.848, E3 +130290.001}
SPL {X  -160.000, Y  +600.731, Z    +0.000, E1   -14.846, E3 +130311.953}
SPL {X  -160.000, Y  +603.404, Z    +0.000, E1   -14.846, E3 +130333.388}
SPL {X  -160.000, Y  +605.923, Z    +0.000, E1   -14.838, E3 +130353.629}
SPL {X  -160.000, Y  +608.492, Z    +0.000, E1   -14.846, E3 +130374.233}
SPL {X  -160.000, Y  +611.345, Z    +0.000, E1   -14.856, E3 +130397.091}
SPL {X  -160.000, Y  +614.087, Z    +0.000, E1   -14.839, E3 +130419.150}
SPL {X  -160.000, Y  +616.566, Z    +0.000, E1   -14.839, E3 +130439.044}
SPL {X  -160.000, Y  +619.350, Z    +0.000, E1   -14.855, E3 +130461.332}
SPL {X  -160.000, Y  +622.198, Z    +0.000, E1   -14.846, E3 +130484.217}
SPL {X  -160.000, Y  +624.642, Z    +0.000, E1   -14.829, E3 +130503.889}
SPL {X  -160.000, Y  +627.119, Z    +0.000, E1   -14.843, E3 +130523.729}
SPL {X  -160.000, Y  +629.682, Z    +0.000, E1   -14.838, E3 +130544.298}
SPL {X  -160.000, Y  +632.223, Z    +0.000, E1   -14.841, E3 +130564.689}
SPL {X  -160.000, Y  +634.941, Z    +0.000, E1   -14.846, E3 +130586.487}
SPL {X  -160.000, Y  +637.723, Z    +0.000, E1   -14.844, E3 +130608.831}
SPL {X  -160.000, Y  +640.315, Z    +0.000, E1   -14.836, E3 +130629.629}
SPL {X  -160.000, Y  +643.085, Z    +0.000, E1   -14.865, E3 +130651.680}
SPL {X  -160.000, Y  +645.845, Z    +0.000, E1   -14.848, E3 +130673.868}
SPL {X  -160.000, Y  +648.229, Z    +0.000, E1   -14.834, E3 +130693.078}
SPL {X  -160.000, Y  +650.656, Z    +0.000, E1   -14.835, E3 +130712.635}
SPL {X  -160.000, Y  +653.134, Z    +0.000, E1   -14.827, E3 +130732.561}
SPL {X  -160.000, Y  +655.670, Z    +0.000, E1   -14.841, E3 +130752.856}
SPL {X  -160.000, Y  +658.349, Z    +0.000, E1   -14.842, E3 +130774.331}
SPL {X  -160.000, Y  +660.936, Z    +0.000, E1   -14.838, E3 +130795.083}
SPL {X  -160.000, Y  +663.567, Z    +0.000, E1   -14.845, E3 +130816.214}
SPL {X  -160.000, Y  +666.216, Z    +0.000, E1   -14.832, E3 +130837.530}
SPL {X  -159.997, Y  +668.731, Z    +0.000, E1   -14.834, E3 +130857.722}
SPL {X  -159.962, Y  +671.176, Z    +0.000, E1   -14.822, E3 +130877.433}
SPL {X  -159.895, Y  +673.507, Z    +0.000, E1   -14.821, E3 +130896.165}
SPL {X  -159.785, Y  +675.985, Z    +0.000, E1   -14.818, E3 +130916.166}
SPL {X  -159.627, Y  +678.622, Z    +0.000, E1   -14.804, E3 +130937.519}
SPL {X  -159.438, Y  +681.094, Z    +0.000, E1   -14.770, E3 +130957.690}
SPL {X  -159.262, Y  +683.054, Z    +0.000, E1   -14.719, E3 +130973.919}
ENDSPLINE

